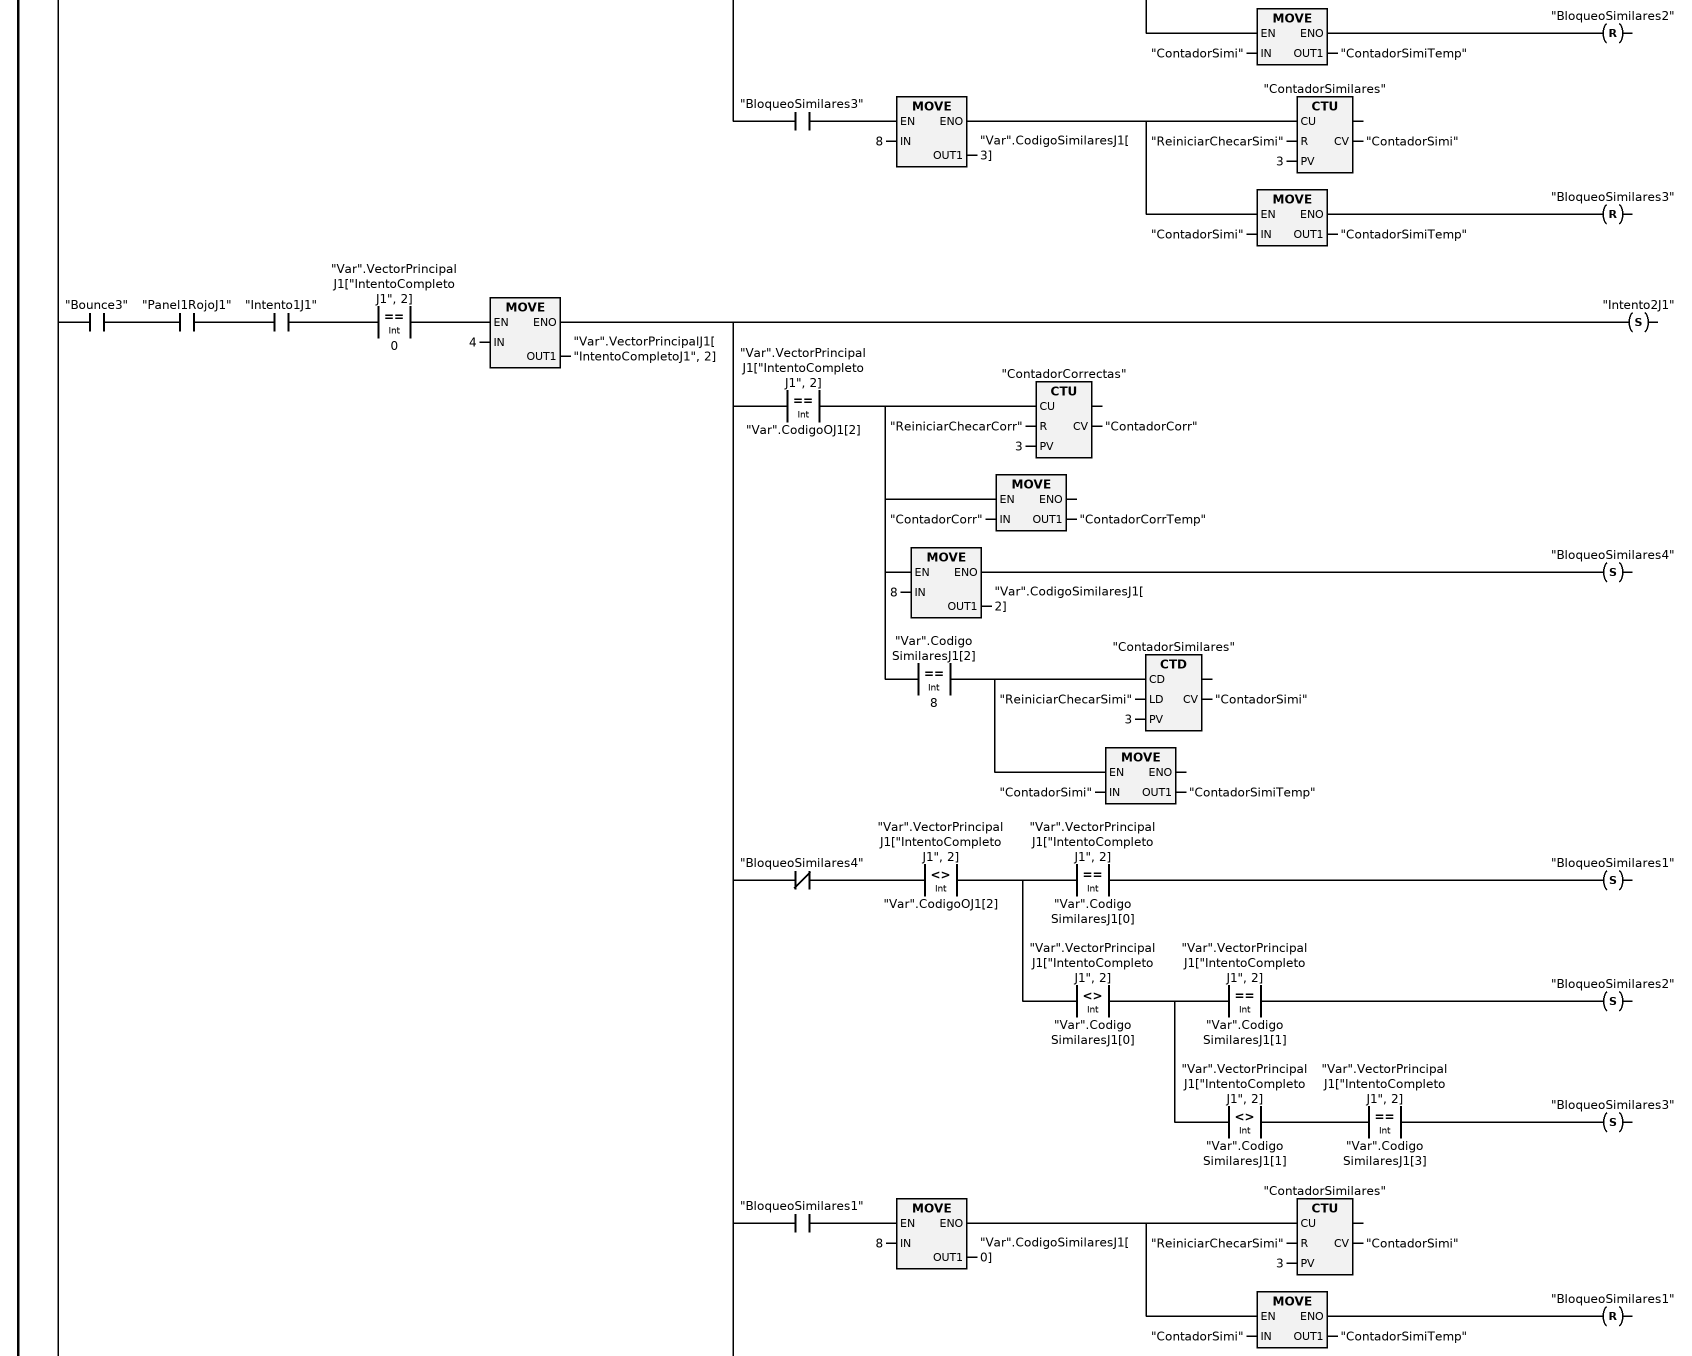
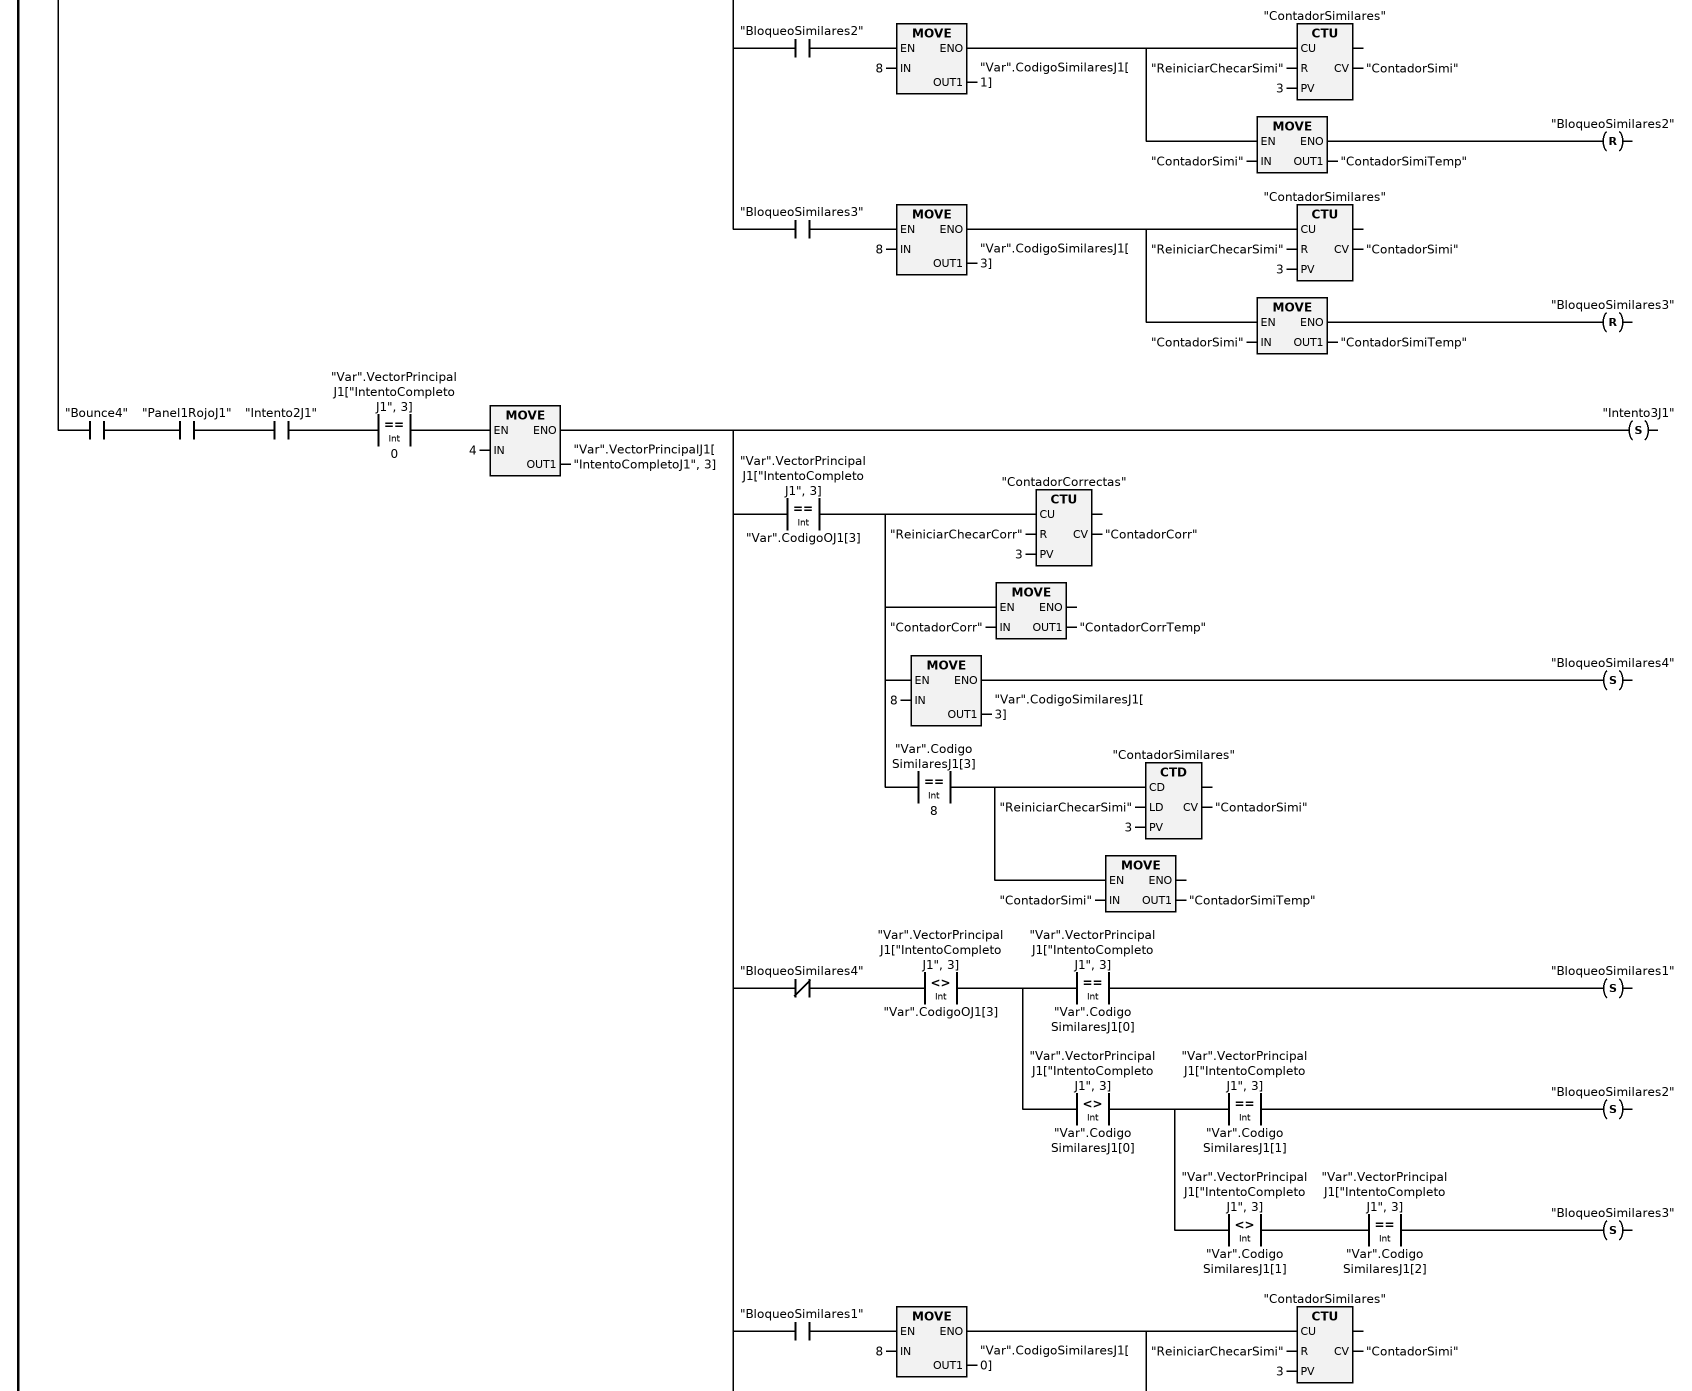
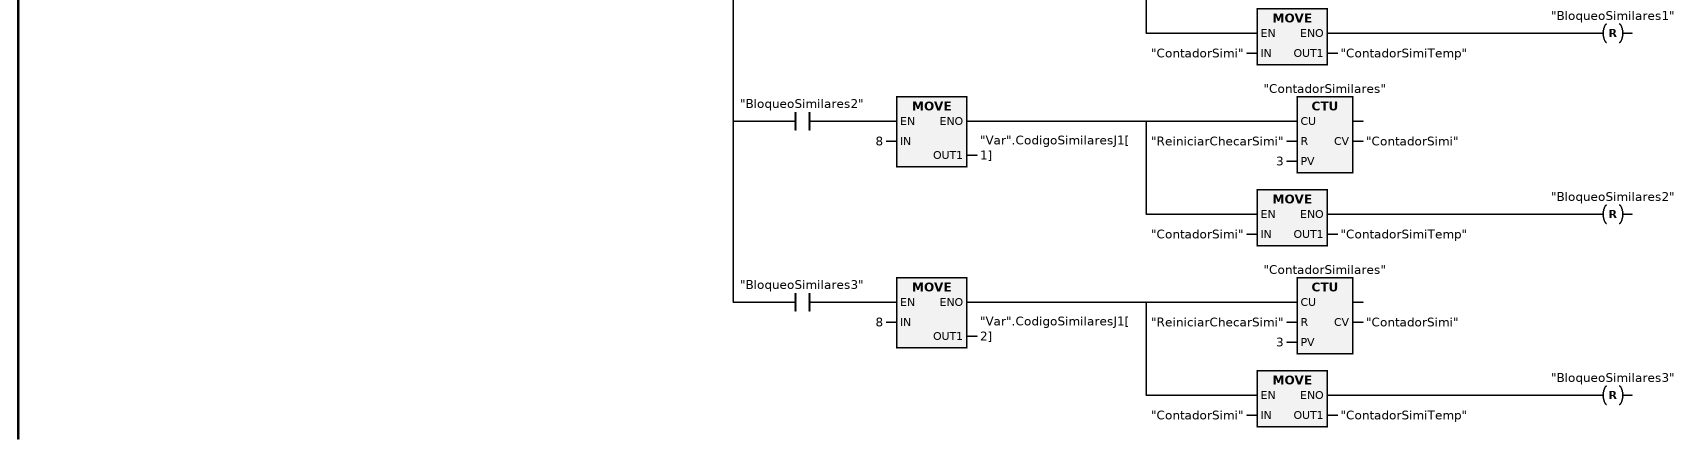
   #_w1 := "Panel1RojoJ1" AND ("Var".VectorPrincipalJ1["IntentoCompletoJ1", 0] = 0) AND "Bounce1";
   IF #_w1 THEN
       "Var".VectorPrincipalJ1["IntentoCompletoJ1", 0] := 4;
       "Var".VectorCorrectas["IntentoCompletoJ1", 0] := 4;
       "Intento0J1" := TRUE;
   END_IF;
   #_w2 := #_w1 AND ("Var".VectorPrincipalJ1["IntentoCompletoJ1", 0] = "Var".CodigoOJ1[0]);
   "ContadorCorrectas".CTU(CU := #_w2, R := "ReiniciarChecarCorr", PV := 3, CV => "ContadorCorr");
   IF #_w2 THEN
       "ContadorCorrTemp" := "ContadorCorr";
       "Var".CodigoSimilaresJ1[0] := 8;
       "BloqueoSimilares4" := TRUE;
   END_IF;
   #_w3 := #_w2 AND ("Var".CodigoSimilaresJ1[0] = 8);
   "ContadorSimilares".CTD(CD := #_w3, LD := "ReiniciarChecarSimi", PV := 3, CV => "ContadorSimi");
   IF #_w3 THEN "ContadorSimiTemp" := "ContadorSimi"; END_IF;
   #_w4 := #_w1 AND NOT "BloqueoSimilares4" AND ("Var".VectorPrincipalJ1["IntentoCompletoJ1", 0] <> "Var".CodigoOJ1[0]);
   IF #_w4 AND ("Var".VectorPrincipalJ1["IntentoCompletoJ1", 0] = "Var".CodigoSimilaresJ1[1]) THEN
       "BloqueoSimilares1" := TRUE;
   END_IF;
   #_w5 := #_w4 AND ("Var".VectorPrincipalJ1["IntentoCompletoJ1", 0] <> "Var".CodigoSimilaresJ1[1]);
   IF #_w5 AND ("Var".VectorPrincipalJ1["IntentoCompletoJ1", 0] = "Var".CodigoSimilaresJ1[2]) THEN
       "BloqueoSimilares2" := TRUE;
   END_IF;
   IF #_w5 AND ("Var".VectorPrincipalJ1["IntentoCompletoJ1", 0] <> "Var".CodigoSimilaresJ1[2]) AND ("Var".VectorPrincipalJ1["IntentoCompletoJ1", 0] = "Var".CodigoSimilaresJ1[3]) THEN
       "BloqueoSimilares3" := TRUE;
   END_IF;
   #_w6 := #_w1 AND "BloqueoSimilares1";
   IF #_w6 THEN "Var".CodigoSimilaresJ1[1] := 8; END_IF;
   "ContadorSimilares".CTU(CU := #_w6, R := "ReiniciarChecarSimi", PV := 3, CV => "ContadorSimi");
   IF #_w6 THEN
       "ContadorSimiTemp" := "ContadorSimi";
       "BloqueoSimilares1" := FALSE;
   END_IF;
   #_w7 := #_w1 AND "BloqueoSimilares2";
   IF #_w7 THEN "Var".CodigoSimilaresJ1[2] := 8; END_IF;
   "ContadorSimilares".CTU(CU := #_w7, R := "ReiniciarChecarSimi", PV := 3, CV => "ContadorSimi");
   IF #_w7 THEN
       "ContadorSimiTemp" := "ContadorSimi";
       "BloqueoSimilares2" := FALSE;
   END_IF;
   #_w8 := #_w1 AND "BloqueoSimilares3";
   IF #_w8 THEN "Var".CodigoSimilaresJ1[3] := 8; END_IF;
   "ContadorSimilares".CTU(CU := #_w8, R := "ReiniciarChecarSimi", PV := 3, CV => "ContadorSimi");
   IF #_w8 THEN
       "ContadorSimiTemp" := "ContadorSimi";
       "BloqueoSimilares3" := FALSE;
   END_IF;
   #_w9 := "Panel1RojoJ1" AND "Bounce2" AND "Panel1RojoJ1" AND "Intento0J1" AND ("Var".VectorPrincipalJ1["IntentoCompletoJ1", 1] = 0);
   IF #_w9 THEN
       "Var".VectorPrincipalJ1["IntentoCompletoJ1", 1] := 4;
       "Intento1J1" := TRUE;
   END_IF;
   #_w10 := #_w9 AND ("Var".VectorPrincipalJ1["IntentoCompletoJ1", 1] = "Var".CodigoOJ1[1]);
   "ContadorCorrectas".CTU(CU := #_w10, R := "ReiniciarChecarCorr", PV := 3, CV => "ContadorCorr");
   IF #_w10 THEN
       "ContadorCorrTemp" := "ContadorCorr";
       "Var".CodigoSimilaresJ1[1] := 8;
       "BloqueoSimilares4" := TRUE;
   END_IF;
   #_w11 := #_w10 AND ("Var".CodigoSimilaresJ1[1] = 8);
   "ContadorSimilares".CTD(CD := #_w11, LD := "ReiniciarChecarSimi", PV := 3, CV => "ContadorSimi");
   IF #_w11 THEN "ContadorSimiTemp" := "ContadorSimi"; END_IF;
   #_w12 := #_w9 AND NOT "BloqueoSimilares4" AND ("Var".VectorPrincipalJ1["IntentoCompletoJ1", 1] <> "Var".CodigoOJ1[1]);
   IF #_w12 AND ("Var".VectorPrincipalJ1["IntentoCompletoJ1", 1] = "Var".CodigoSimilaresJ1[0]) THEN
       "BloqueoSimilares1" := TRUE;
   END_IF;
   #_w13 := #_w12 AND ("Var".VectorPrincipalJ1["IntentoCompletoJ1", 1] <> "Var".CodigoSimilaresJ1[0]);
   IF #_w13 AND ("Var".VectorPrincipalJ1["IntentoCompletoJ1", 1] = "Var".CodigoSimilaresJ1[2]) THEN
       "BloqueoSimilares2" := TRUE;
   END_IF;
   IF #_w13 AND ("Var".VectorPrincipalJ1["IntentoCompletoJ1", 1] <> "Var".CodigoSimilaresJ1[2]) AND ("Var".VectorPrincipalJ1["IntentoCompletoJ1", 1] = "Var".CodigoSimilaresJ1[3]) THEN
       "BloqueoSimilares3" := TRUE;
   END_IF;
   #_w14 := #_w9 AND "BloqueoSimilares1";
   IF #_w14 THEN "Var".CodigoSimilaresJ1[0] := 8; END_IF;
   "ContadorSimilares".CTU(CU := #_w14, R := "ReiniciarChecarSimi", PV := 3, CV => "ContadorSimi");
   IF #_w14 THEN
       "ContadorSimiTemp" := "ContadorSimi";
       "BloqueoSimilares1" := FALSE;
   END_IF;
   #_w15 := #_w9 AND "BloqueoSimilares2";
   IF #_w15 THEN "Var".CodigoSimilaresJ1[2] := 8; END_IF;
   "ContadorSimilares".CTU(CU := #_w15, R := "ReiniciarChecarSimi", PV := 3, CV => "ContadorSimi");
   IF #_w15 THEN
       "ContadorSimiTemp" := "ContadorSimi";
       "BloqueoSimilares2" := FALSE;
   END_IF;
   #_w16 := #_w9 AND "BloqueoSimilares3";
   IF #_w16 THEN "Var".CodigoSimilaresJ1[3] := 8; END_IF;
   "ContadorSimilares".CTU(CU := #_w16, R := "ReiniciarChecarSimi", PV := 3, CV => "ContadorSimi");
   IF #_w16 THEN
       "ContadorSimiTemp" := "ContadorSimi";
       "BloqueoSimilares3" := FALSE;
   END_IF;
   #_w17 := "Panel1RojoJ1" AND "Bounce3" AND "Panel1RojoJ1" AND "Intento1J1" AND ("Var".VectorPrincipalJ1["IntentoCompletoJ1", 2] = 0);
   IF #_w17 THEN
       "Var".VectorPrincipalJ1["IntentoCompletoJ1", 2] := 4;
       "Intento2J1" := TRUE;
   END_IF;
   #_w18 := #_w17 AND ("Var".VectorPrincipalJ1["IntentoCompletoJ1", 2] = "Var".CodigoOJ1[2]);
   "ContadorCorrectas".CTU(CU := #_w18, R := "ReiniciarChecarCorr", PV := 3, CV => "ContadorCorr");
   IF #_w18 THEN
       "ContadorCorrTemp" := "ContadorCorr";
       "Var".CodigoSimilaresJ1[2] := 8;
       "BloqueoSimilares4" := TRUE;
   END_IF;
   #_w19 := #_w18 AND ("Var".CodigoSimilaresJ1[2] = 8);
   "ContadorSimilares".CTD(CD := #_w19, LD := "ReiniciarChecarSimi", PV := 3, CV => "ContadorSimi");
   IF #_w19 THEN "ContadorSimiTemp" := "ContadorSimi"; END_IF;
   #_w20 := #_w17 AND NOT "BloqueoSimilares4" AND ("Var".VectorPrincipalJ1["IntentoCompletoJ1", 2] <> "Var".CodigoOJ1[2]);
   IF #_w20 AND ("Var".VectorPrincipalJ1["IntentoCompletoJ1", 2] = "Var".CodigoSimilaresJ1[0]) THEN
       "BloqueoSimilares1" := TRUE;
   END_IF;
   #_w21 := #_w20 AND ("Var".VectorPrincipalJ1["IntentoCompletoJ1", 2] <> "Var".CodigoSimilaresJ1[0]);
   IF #_w21 AND ("Var".VectorPrincipalJ1["IntentoCompletoJ1", 2] = "Var".CodigoSimilaresJ1[1]) THEN
       "BloqueoSimilares2" := TRUE;
   END_IF;
   IF #_w21 AND ("Var".VectorPrincipalJ1["IntentoCompletoJ1", 2] <> "Var".CodigoSimilaresJ1[1]) AND ("Var".VectorPrincipalJ1["IntentoCompletoJ1", 2] = "Var".CodigoSimilaresJ1[3]) THEN
       "BloqueoSimilares3" := TRUE;
   END_IF;
   #_w22 := #_w17 AND "BloqueoSimilares1";
   IF #_w22 THEN "Var".CodigoSimilaresJ1[0] := 8; END_IF;
   "ContadorSimilares".CTU(CU := #_w22, R := "ReiniciarChecarSimi", PV := 3, CV => "ContadorSimi");
   IF #_w22 THEN
       "ContadorSimiTemp" := "ContadorSimi";
       "BloqueoSimilares1" := FALSE;
   END_IF;
   #_w23 := #_w17 AND "BloqueoSimilares2";
   IF #_w23 THEN "Var".CodigoSimilaresJ1[1] := 8; END_IF;
   "ContadorSimilares".CTU(CU := #_w23, R := "ReiniciarChecarSimi", PV := 3, CV => "ContadorSimi");
   IF #_w23 THEN
       "ContadorSimiTemp" := "ContadorSimi";
       "BloqueoSimilares2" := FALSE;
   END_IF;
   #_w24 := #_w17 AND "BloqueoSimilares3";
   IF #_w24 THEN "Var".CodigoSimilaresJ1[3] := 8; END_IF;
   "ContadorSimilares".CTU(CU := #_w24, R := "ReiniciarChecarSimi", PV := 3, CV => "ContadorSimi");
   IF #_w24 THEN
       "ContadorSimiTemp" := "ContadorSimi";
       "BloqueoSimilares3" := FALSE;
   END_IF;
   #_w25 := "Panel1RojoJ1" AND "Bounce4" AND "Panel1RojoJ1" AND "Intento2J1" AND ("Var".VectorPrincipalJ1["IntentoCompletoJ1", 3] = 0);
   IF #_w25 THEN
       "Var".VectorPrincipalJ1["IntentoCompletoJ1", 3] := 4;
       "Intento3J1" := TRUE;
   END_IF;
   #_w26 := #_w25 AND ("Var".VectorPrincipalJ1["IntentoCompletoJ1", 3] = "Var".CodigoOJ1[3]);
   "ContadorCorrectas".CTU(CU := #_w26, R := "ReiniciarChecarCorr", PV := 3, CV => "ContadorCorr");
   IF #_w26 THEN
       "ContadorCorrTemp" := "ContadorCorr";
       "Var".CodigoSimilaresJ1[3] := 8;
       "BloqueoSimilares4" := TRUE;
   END_IF;
   #_w27 := #_w26 AND ("Var".CodigoSimilaresJ1[3] = 8);
   "ContadorSimilares".CTD(CD := #_w27, LD := "ReiniciarChecarSimi", PV := 3, CV => "ContadorSimi");
   IF #_w27 THEN "ContadorSimiTemp" := "ContadorSimi"; END_IF;
   #_w28 := #_w25 AND NOT "BloqueoSimilares4" AND ("Var".VectorPrincipalJ1["IntentoCompletoJ1", 3] <> "Var".CodigoOJ1[3]);
   IF #_w28 AND ("Var".VectorPrincipalJ1["IntentoCompletoJ1", 3] = "Var".CodigoSimilaresJ1[0]) THEN
       "BloqueoSimilares1" := TRUE;
   END_IF;
   #_w29 := #_w28 AND ("Var".VectorPrincipalJ1["IntentoCompletoJ1", 3] <> "Var".CodigoSimilaresJ1[0]);
   IF #_w29 AND ("Var".VectorPrincipalJ1["IntentoCompletoJ1", 3] = "Var".CodigoSimilaresJ1[1]) THEN
       "BloqueoSimilares2" := TRUE;
   END_IF;
   IF #_w29 AND ("Var".VectorPrincipalJ1["IntentoCompletoJ1", 3] <> "Var".CodigoSimilaresJ1[1]) AND ("Var".VectorPrincipalJ1["IntentoCompletoJ1", 3] = "Var".CodigoSimilaresJ1[2]) THEN
       "BloqueoSimilares3" := TRUE;
   END_IF;
   #_w30 := #_w25 AND "BloqueoSimilares1";
   IF #_w30 THEN "Var".CodigoSimilaresJ1[0] := 8; END_IF;
   "ContadorSimilares".CTU(CU := #_w30, R := "ReiniciarChecarSimi", PV := 3, CV => "ContadorSimi");
   IF #_w30 THEN
       "ContadorSimiTemp" := "ContadorSimi";
       "BloqueoSimilares1" := FALSE;
   END_IF;
   #_w31 := #_w25 AND "BloqueoSimilares2";
   IF #_w31 THEN "Var".CodigoSimilaresJ1[1] := 8; END_IF;
   "ContadorSimilares".CTU(CU := #_w31, R := "ReiniciarChecarSimi", PV := 3, CV => "ContadorSimi");
   IF #_w31 THEN
       "ContadorSimiTemp" := "ContadorSimi";
       "BloqueoSimilares2" := FALSE;
   END_IF;
   #_w32 := #_w25 AND "BloqueoSimilares3";
   IF #_w32 THEN "Var".CodigoSimilaresJ1[2] := 8; END_IF;
   "ContadorSimilares".CTU(CU := #_w32, R := "ReiniciarChecarSimi", PV := 3, CV => "ContadorSimi");
   IF #_w32 THEN
       "ContadorSimiTemp" := "ContadorSimi";
       "BloqueoSimilares3" := FALSE;
   END_IF;
END_REGION

REGION Network 10: Azul
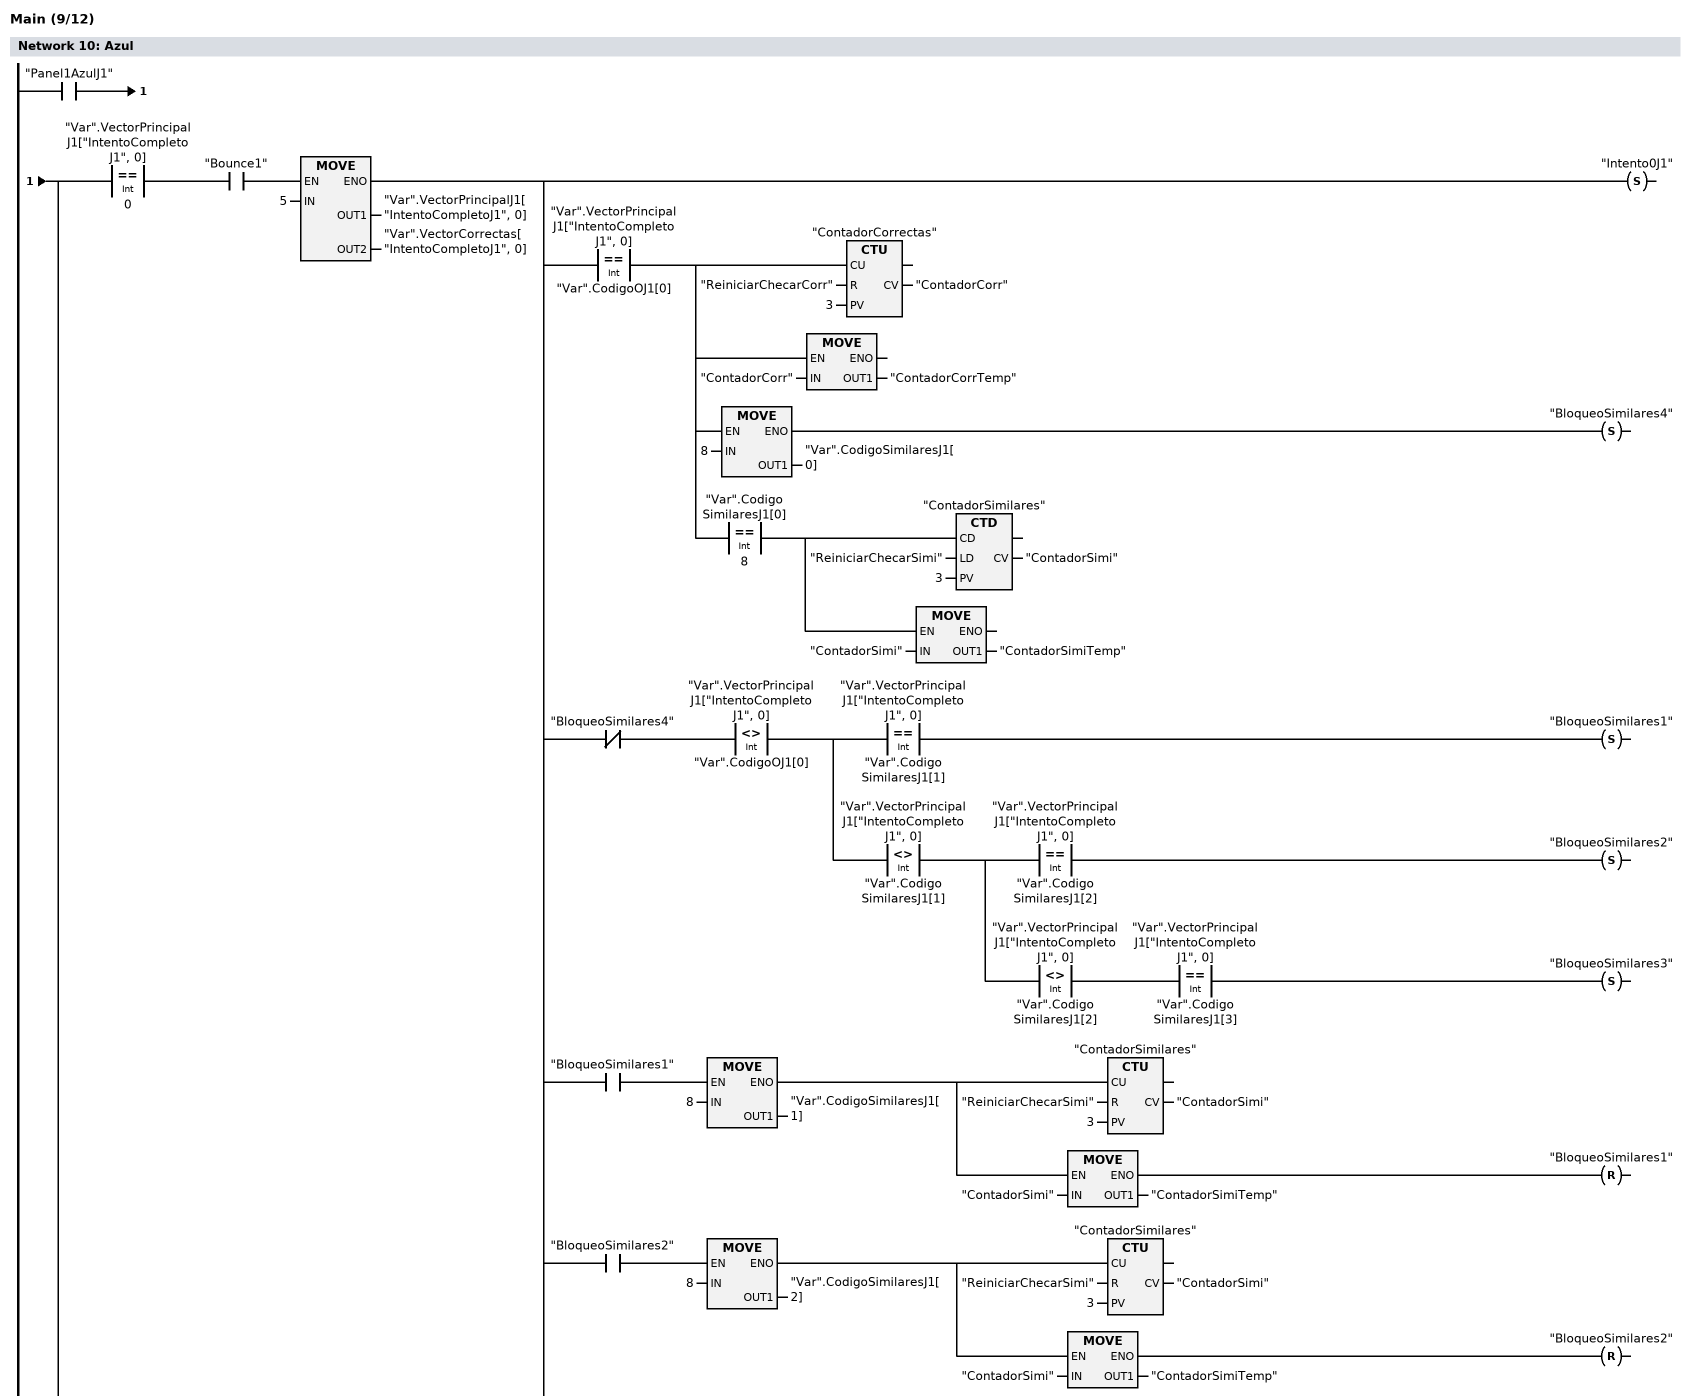
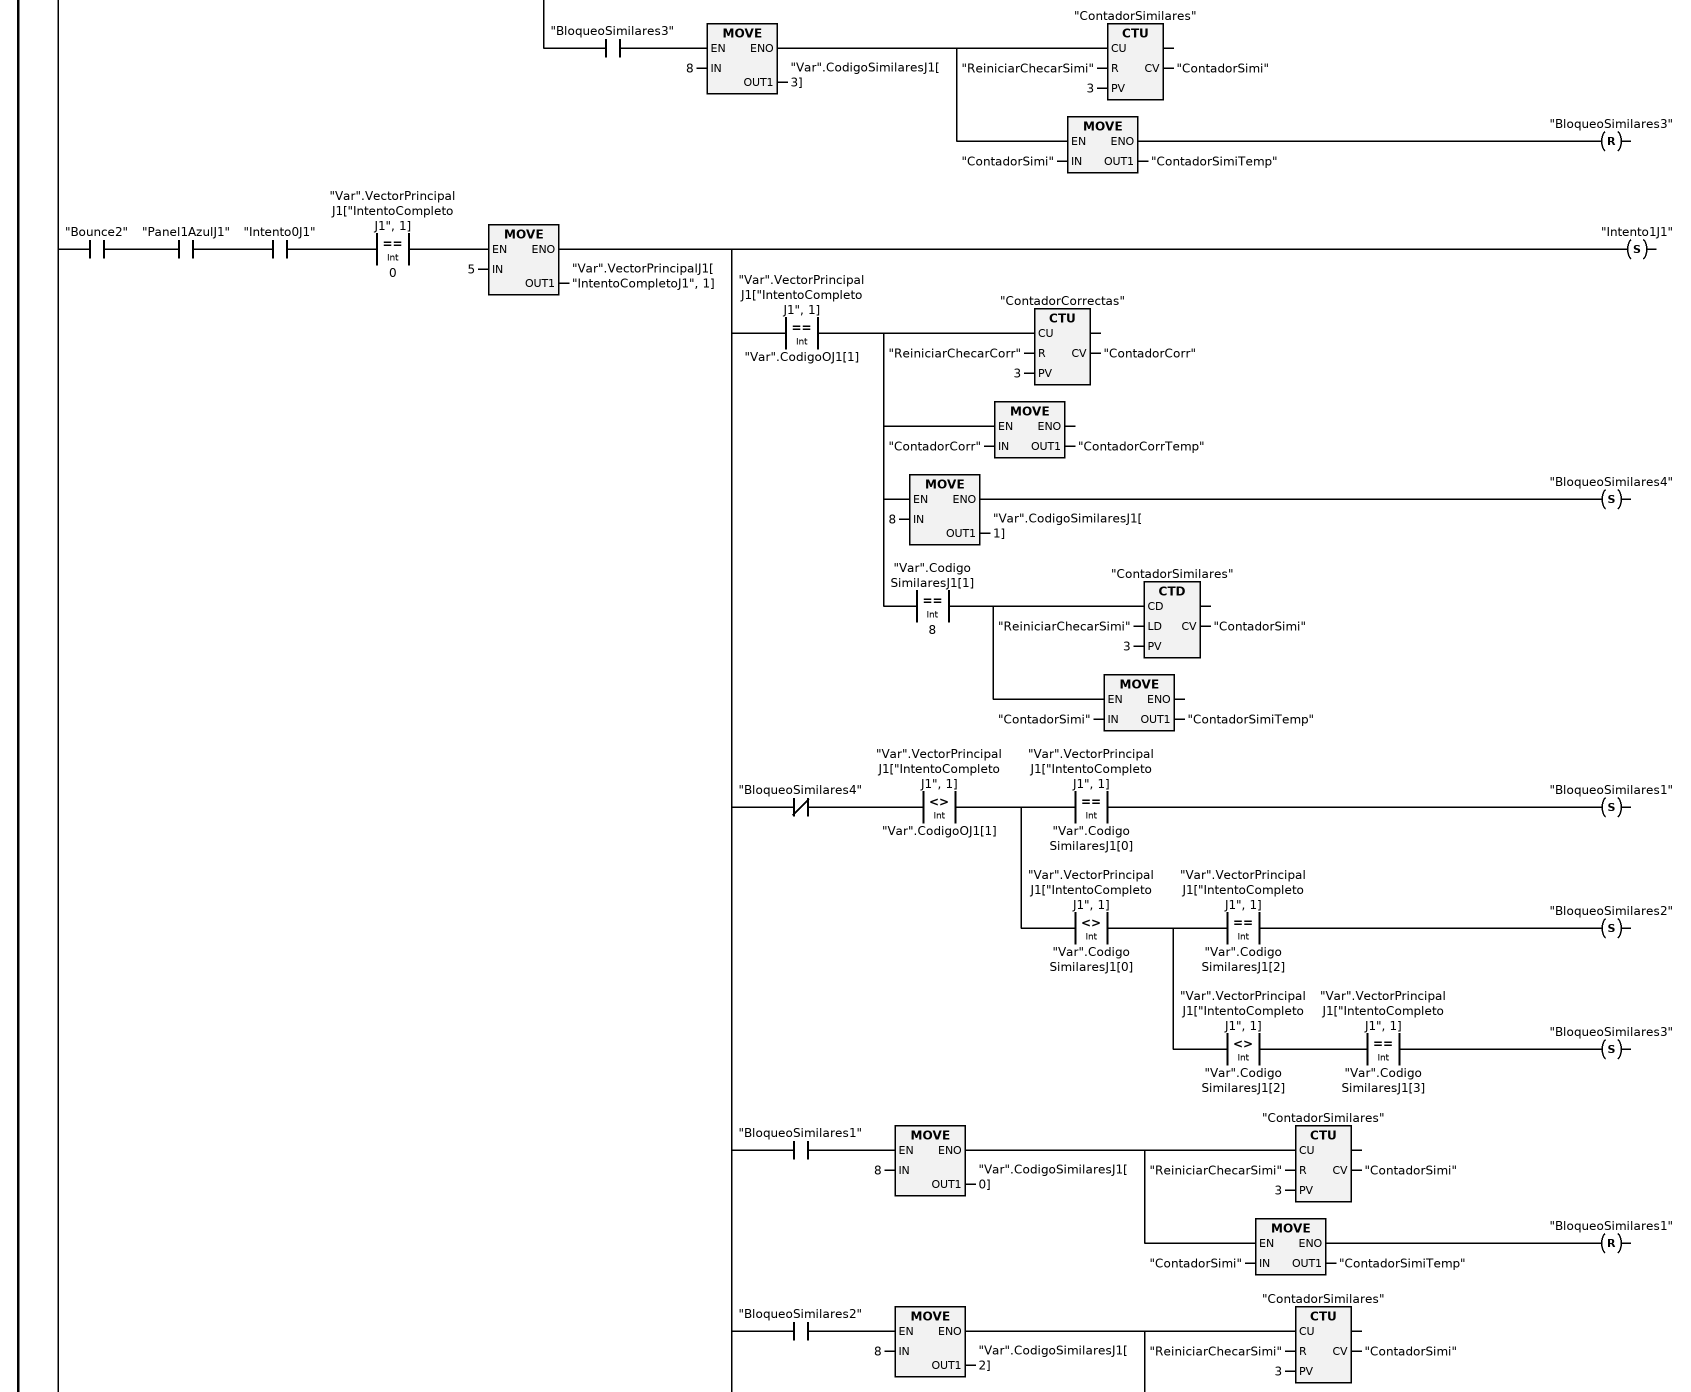
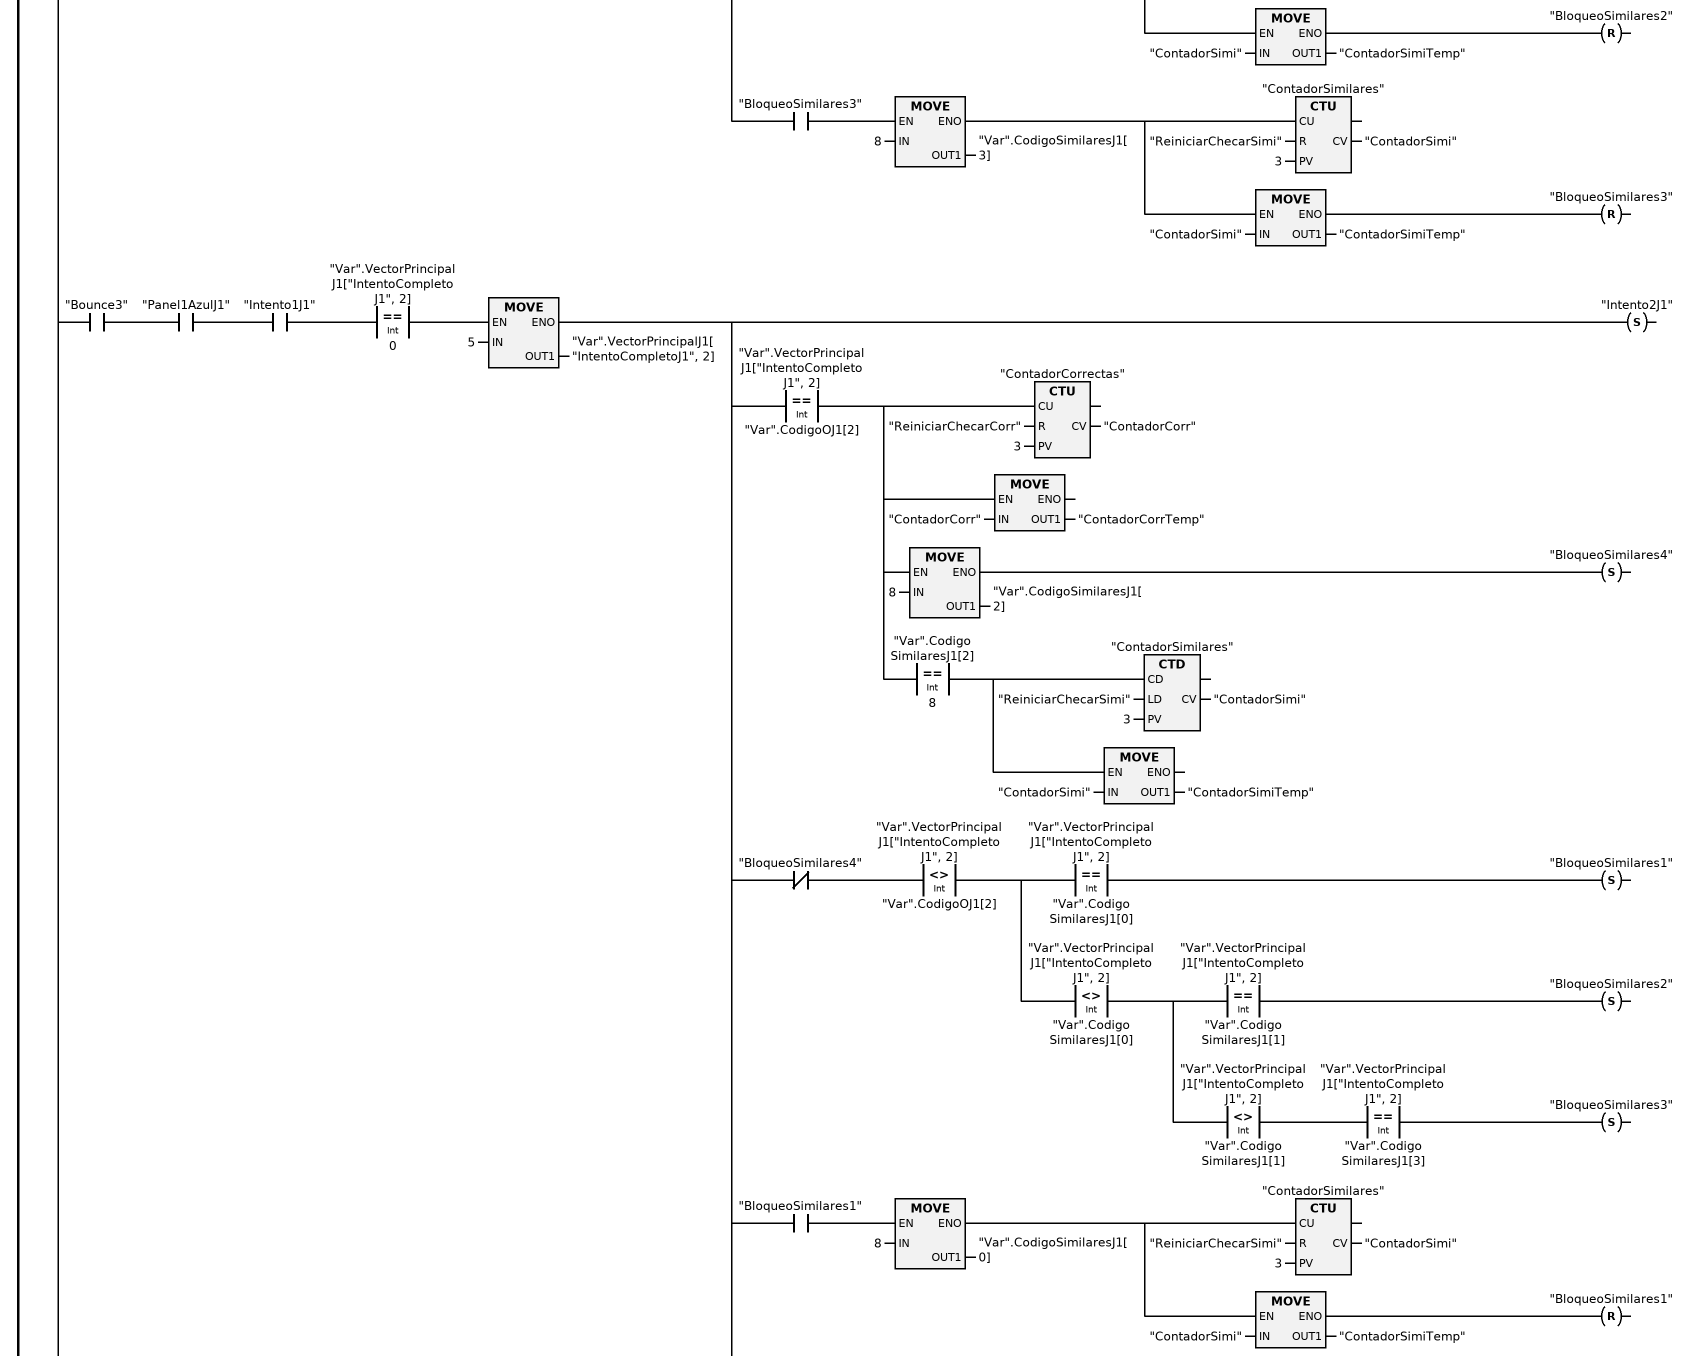
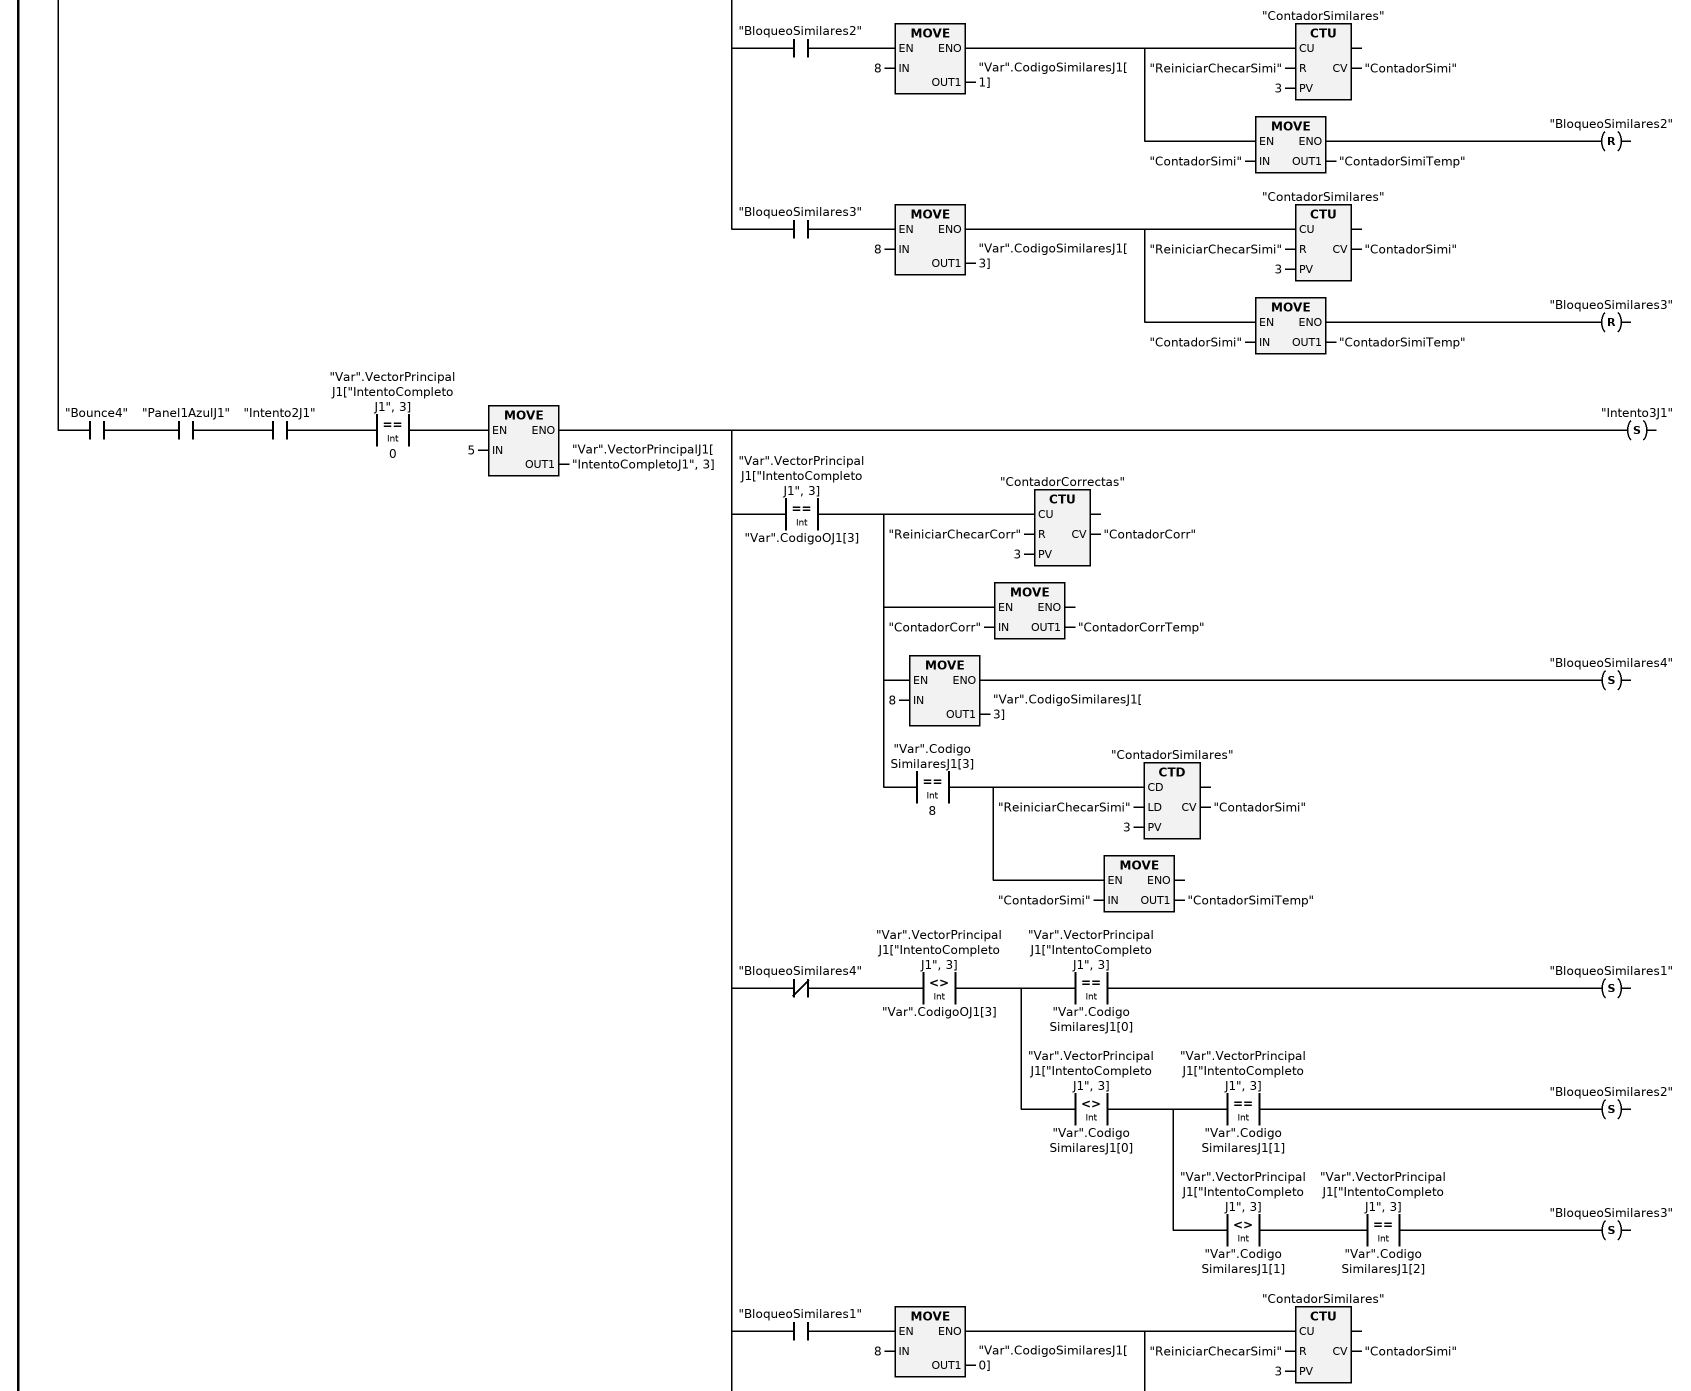
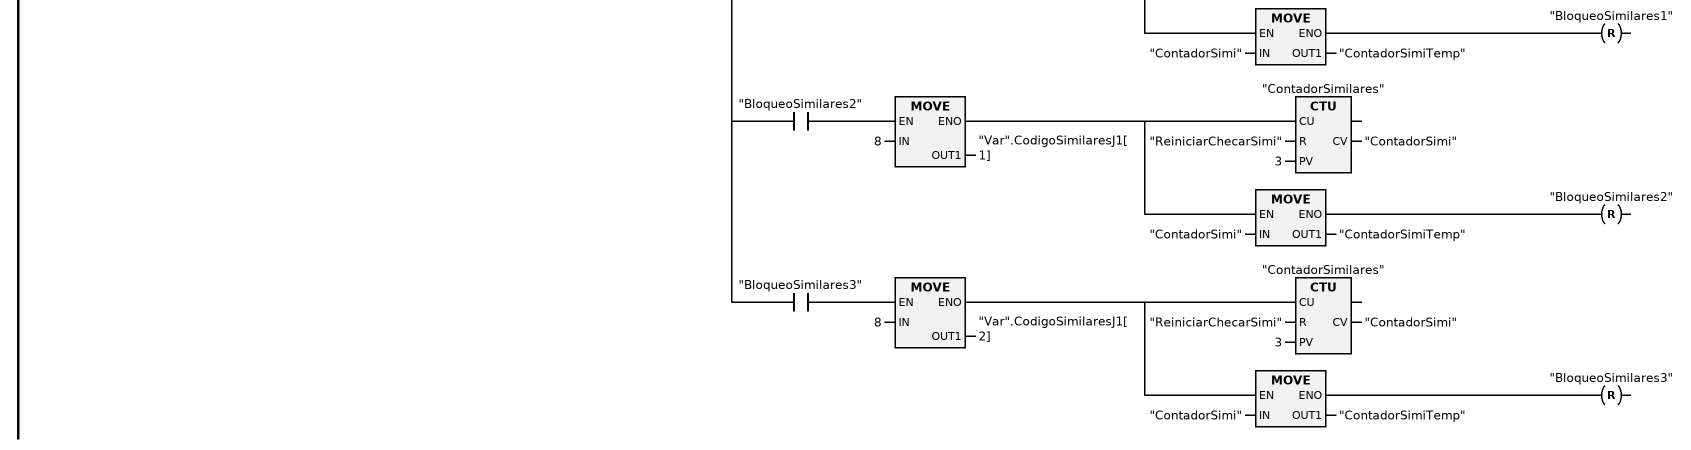
   #_w1 := "Panel1AzulJ1" AND ("Var".VectorPrincipalJ1["IntentoCompletoJ1", 0] = 0) AND "Bounce1";
   IF #_w1 THEN
       "Var".VectorPrincipalJ1["IntentoCompletoJ1", 0] := 5;
       "Var".VectorCorrectas["IntentoCompletoJ1", 0] := 5;
       "Intento0J1" := TRUE;
   END_IF;
   #_w2 := #_w1 AND ("Var".VectorPrincipalJ1["IntentoCompletoJ1", 0] = "Var".CodigoOJ1[0]);
   "ContadorCorrectas".CTU(CU := #_w2, R := "ReiniciarChecarCorr", PV := 3, CV => "ContadorCorr");
   IF #_w2 THEN
       "ContadorCorrTemp" := "ContadorCorr";
       "Var".CodigoSimilaresJ1[0] := 8;
       "BloqueoSimilares4" := TRUE;
   END_IF;
   #_w3 := #_w2 AND ("Var".CodigoSimilaresJ1[0] = 8);
   "ContadorSimilares".CTD(CD := #_w3, LD := "ReiniciarChecarSimi", PV := 3, CV => "ContadorSimi");
   IF #_w3 THEN "ContadorSimiTemp" := "ContadorSimi"; END_IF;
   #_w4 := #_w1 AND NOT "BloqueoSimilares4" AND ("Var".VectorPrincipalJ1["IntentoCompletoJ1", 0] <> "Var".CodigoOJ1[0]);
   IF #_w4 AND ("Var".VectorPrincipalJ1["IntentoCompletoJ1", 0] = "Var".CodigoSimilaresJ1[1]) THEN
       "BloqueoSimilares1" := TRUE;
   END_IF;
   #_w5 := #_w4 AND ("Var".VectorPrincipalJ1["IntentoCompletoJ1", 0] <> "Var".CodigoSimilaresJ1[1]);
   IF #_w5 AND ("Var".VectorPrincipalJ1["IntentoCompletoJ1", 0] = "Var".CodigoSimilaresJ1[2]) THEN
       "BloqueoSimilares2" := TRUE;
   END_IF;
   IF #_w5 AND ("Var".VectorPrincipalJ1["IntentoCompletoJ1", 0] <> "Var".CodigoSimilaresJ1[2]) AND ("Var".VectorPrincipalJ1["IntentoCompletoJ1", 0] = "Var".CodigoSimilaresJ1[3]) THEN
       "BloqueoSimilares3" := TRUE;
   END_IF;
   #_w6 := #_w1 AND "BloqueoSimilares1";
   IF #_w6 THEN "Var".CodigoSimilaresJ1[1] := 8; END_IF;
   "ContadorSimilares".CTU(CU := #_w6, R := "ReiniciarChecarSimi", PV := 3, CV => "ContadorSimi");
   IF #_w6 THEN
       "ContadorSimiTemp" := "ContadorSimi";
       "BloqueoSimilares1" := FALSE;
   END_IF;
   #_w7 := #_w1 AND "BloqueoSimilares2";
   IF #_w7 THEN "Var".CodigoSimilaresJ1[2] := 8; END_IF;
   "ContadorSimilares".CTU(CU := #_w7, R := "ReiniciarChecarSimi", PV := 3, CV => "ContadorSimi");
   IF #_w7 THEN
       "ContadorSimiTemp" := "ContadorSimi";
       "BloqueoSimilares2" := FALSE;
   END_IF;
   #_w8 := #_w1 AND "BloqueoSimilares3";
   IF #_w8 THEN "Var".CodigoSimilaresJ1[3] := 8; END_IF;
   "ContadorSimilares".CTU(CU := #_w8, R := "ReiniciarChecarSimi", PV := 3, CV => "ContadorSimi");
   IF #_w8 THEN
       "ContadorSimiTemp" := "ContadorSimi";
       "BloqueoSimilares3" := FALSE;
   END_IF;
   #_w9 := "Panel1AzulJ1" AND "Bounce2" AND "Panel1AzulJ1" AND "Intento0J1" AND ("Var".VectorPrincipalJ1["IntentoCompletoJ1", 1] = 0);
   IF #_w9 THEN
       "Var".VectorPrincipalJ1["IntentoCompletoJ1", 1] := 5;
       "Intento1J1" := TRUE;
   END_IF;
   #_w10 := #_w9 AND ("Var".VectorPrincipalJ1["IntentoCompletoJ1", 1] = "Var".CodigoOJ1[1]);
   "ContadorCorrectas".CTU(CU := #_w10, R := "ReiniciarChecarCorr", PV := 3, CV => "ContadorCorr");
   IF #_w10 THEN
       "ContadorCorrTemp" := "ContadorCorr";
       "Var".CodigoSimilaresJ1[1] := 8;
       "BloqueoSimilares4" := TRUE;
   END_IF;
   #_w11 := #_w10 AND ("Var".CodigoSimilaresJ1[1] = 8);
   "ContadorSimilares".CTD(CD := #_w11, LD := "ReiniciarChecarSimi", PV := 3, CV => "ContadorSimi");
   IF #_w11 THEN "ContadorSimiTemp" := "ContadorSimi"; END_IF;
   #_w12 := #_w9 AND NOT "BloqueoSimilares4" AND ("Var".VectorPrincipalJ1["IntentoCompletoJ1", 1] <> "Var".CodigoOJ1[1]);
   IF #_w12 AND ("Var".VectorPrincipalJ1["IntentoCompletoJ1", 1] = "Var".CodigoSimilaresJ1[0]) THEN
       "BloqueoSimilares1" := TRUE;
   END_IF;
   #_w13 := #_w12 AND ("Var".VectorPrincipalJ1["IntentoCompletoJ1", 1] <> "Var".CodigoSimilaresJ1[0]);
   IF #_w13 AND ("Var".VectorPrincipalJ1["IntentoCompletoJ1", 1] = "Var".CodigoSimilaresJ1[2]) THEN
       "BloqueoSimilares2" := TRUE;
   END_IF;
   IF #_w13 AND ("Var".VectorPrincipalJ1["IntentoCompletoJ1", 1] <> "Var".CodigoSimilaresJ1[2]) AND ("Var".VectorPrincipalJ1["IntentoCompletoJ1", 1] = "Var".CodigoSimilaresJ1[3]) THEN
       "BloqueoSimilares3" := TRUE;
   END_IF;
   #_w14 := #_w9 AND "BloqueoSimilares1";
   IF #_w14 THEN "Var".CodigoSimilaresJ1[0] := 8; END_IF;
   "ContadorSimilares".CTU(CU := #_w14, R := "ReiniciarChecarSimi", PV := 3, CV => "ContadorSimi");
   IF #_w14 THEN
       "ContadorSimiTemp" := "ContadorSimi";
       "BloqueoSimilares1" := FALSE;
   END_IF;
   #_w15 := #_w9 AND "BloqueoSimilares2";
   IF #_w15 THEN "Var".CodigoSimilaresJ1[2] := 8; END_IF;
   "ContadorSimilares".CTU(CU := #_w15, R := "ReiniciarChecarSimi", PV := 3, CV => "ContadorSimi");
   IF #_w15 THEN
       "ContadorSimiTemp" := "ContadorSimi";
       "BloqueoSimilares2" := FALSE;
   END_IF;
   #_w16 := #_w9 AND "BloqueoSimilares3";
   IF #_w16 THEN "Var".CodigoSimilaresJ1[3] := 8; END_IF;
   "ContadorSimilares".CTU(CU := #_w16, R := "ReiniciarChecarSimi", PV := 3, CV => "ContadorSimi");
   IF #_w16 THEN
       "ContadorSimiTemp" := "ContadorSimi";
       "BloqueoSimilares3" := FALSE;
   END_IF;
   #_w17 := "Panel1AzulJ1" AND "Bounce3" AND "Panel1AzulJ1" AND "Intento1J1" AND ("Var".VectorPrincipalJ1["IntentoCompletoJ1", 2] = 0);
   IF #_w17 THEN
       "Var".VectorPrincipalJ1["IntentoCompletoJ1", 2] := 5;
       "Intento2J1" := TRUE;
   END_IF;
   #_w18 := #_w17 AND ("Var".VectorPrincipalJ1["IntentoCompletoJ1", 2] = "Var".CodigoOJ1[2]);
   "ContadorCorrectas".CTU(CU := #_w18, R := "ReiniciarChecarCorr", PV := 3, CV => "ContadorCorr");
   IF #_w18 THEN
       "ContadorCorrTemp" := "ContadorCorr";
       "Var".CodigoSimilaresJ1[2] := 8;
       "BloqueoSimilares4" := TRUE;
   END_IF;
   #_w19 := #_w18 AND ("Var".CodigoSimilaresJ1[2] = 8);
   "ContadorSimilares".CTD(CD := #_w19, LD := "ReiniciarChecarSimi", PV := 3, CV => "ContadorSimi");
   IF #_w19 THEN "ContadorSimiTemp" := "ContadorSimi"; END_IF;
   #_w20 := #_w17 AND NOT "BloqueoSimilares4" AND ("Var".VectorPrincipalJ1["IntentoCompletoJ1", 2] <> "Var".CodigoOJ1[2]);
   IF #_w20 AND ("Var".VectorPrincipalJ1["IntentoCompletoJ1", 2] = "Var".CodigoSimilaresJ1[0]) THEN
       "BloqueoSimilares1" := TRUE;
   END_IF;
   #_w21 := #_w20 AND ("Var".VectorPrincipalJ1["IntentoCompletoJ1", 2] <> "Var".CodigoSimilaresJ1[0]);
   IF #_w21 AND ("Var".VectorPrincipalJ1["IntentoCompletoJ1", 2] = "Var".CodigoSimilaresJ1[1]) THEN
       "BloqueoSimilares2" := TRUE;
   END_IF;
   IF #_w21 AND ("Var".VectorPrincipalJ1["IntentoCompletoJ1", 2] <> "Var".CodigoSimilaresJ1[1]) AND ("Var".VectorPrincipalJ1["IntentoCompletoJ1", 2] = "Var".CodigoSimilaresJ1[3]) THEN
       "BloqueoSimilares3" := TRUE;
   END_IF;
   #_w22 := #_w17 AND "BloqueoSimilares1";
   IF #_w22 THEN "Var".CodigoSimilaresJ1[0] := 8; END_IF;
   "ContadorSimilares".CTU(CU := #_w22, R := "ReiniciarChecarSimi", PV := 3, CV => "ContadorSimi");
   IF #_w22 THEN
       "ContadorSimiTemp" := "ContadorSimi";
       "BloqueoSimilares1" := FALSE;
   END_IF;
   #_w23 := #_w17 AND "BloqueoSimilares2";
   IF #_w23 THEN "Var".CodigoSimilaresJ1[1] := 8; END_IF;
   "ContadorSimilares".CTU(CU := #_w23, R := "ReiniciarChecarSimi", PV := 3, CV => "ContadorSimi");
   IF #_w23 THEN
       "ContadorSimiTemp" := "ContadorSimi";
       "BloqueoSimilares2" := FALSE;
   END_IF;
   #_w24 := #_w17 AND "BloqueoSimilares3";
   IF #_w24 THEN "Var".CodigoSimilaresJ1[3] := 8; END_IF;
   "ContadorSimilares".CTU(CU := #_w24, R := "ReiniciarChecarSimi", PV := 3, CV => "ContadorSimi");
   IF #_w24 THEN
       "ContadorSimiTemp" := "ContadorSimi";
       "BloqueoSimilares3" := FALSE;
   END_IF;
   #_w25 := "Panel1AzulJ1" AND "Bounce4" AND "Panel1AzulJ1" AND "Intento2J1" AND ("Var".VectorPrincipalJ1["IntentoCompletoJ1", 3] = 0);
   IF #_w25 THEN
       "Var".VectorPrincipalJ1["IntentoCompletoJ1", 3] := 5;
       "Intento3J1" := TRUE;
   END_IF;
   #_w26 := #_w25 AND ("Var".VectorPrincipalJ1["IntentoCompletoJ1", 3] = "Var".CodigoOJ1[3]);
   "ContadorCorrectas".CTU(CU := #_w26, R := "ReiniciarChecarCorr", PV := 3, CV => "ContadorCorr");
   IF #_w26 THEN
       "ContadorCorrTemp" := "ContadorCorr";
       "Var".CodigoSimilaresJ1[3] := 8;
       "BloqueoSimilares4" := TRUE;
   END_IF;
   #_w27 := #_w26 AND ("Var".CodigoSimilaresJ1[3] = 8);
   "ContadorSimilares".CTD(CD := #_w27, LD := "ReiniciarChecarSimi", PV := 3, CV => "ContadorSimi");
   IF #_w27 THEN "ContadorSimiTemp" := "ContadorSimi"; END_IF;
   #_w28 := #_w25 AND NOT "BloqueoSimilares4" AND ("Var".VectorPrincipalJ1["IntentoCompletoJ1", 3] <> "Var".CodigoOJ1[3]);
   IF #_w28 AND ("Var".VectorPrincipalJ1["IntentoCompletoJ1", 3] = "Var".CodigoSimilaresJ1[0]) THEN
       "BloqueoSimilares1" := TRUE;
   END_IF;
   #_w29 := #_w28 AND ("Var".VectorPrincipalJ1["IntentoCompletoJ1", 3] <> "Var".CodigoSimilaresJ1[0]);
   IF #_w29 AND ("Var".VectorPrincipalJ1["IntentoCompletoJ1", 3] = "Var".CodigoSimilaresJ1[1]) THEN
       "BloqueoSimilares2" := TRUE;
   END_IF;
   IF #_w29 AND ("Var".VectorPrincipalJ1["IntentoCompletoJ1", 3] <> "Var".CodigoSimilaresJ1[1]) AND ("Var".VectorPrincipalJ1["IntentoCompletoJ1", 3] = "Var".CodigoSimilaresJ1[2]) THEN
       "BloqueoSimilares3" := TRUE;
   END_IF;
   #_w30 := #_w25 AND "BloqueoSimilares1";
   IF #_w30 THEN "Var".CodigoSimilaresJ1[0] := 8; END_IF;
   "ContadorSimilares".CTU(CU := #_w30, R := "ReiniciarChecarSimi", PV := 3, CV => "ContadorSimi");
   IF #_w30 THEN
       "ContadorSimiTemp" := "ContadorSimi";
       "BloqueoSimilares1" := FALSE;
   END_IF;
   #_w31 := #_w25 AND "BloqueoSimilares2";
   IF #_w31 THEN "Var".CodigoSimilaresJ1[1] := 8; END_IF;
   "ContadorSimilares".CTU(CU := #_w31, R := "ReiniciarChecarSimi", PV := 3, CV => "ContadorSimi");
   IF #_w31 THEN
       "ContadorSimiTemp" := "ContadorSimi";
       "BloqueoSimilares2" := FALSE;
   END_IF;
   #_w32 := #_w25 AND "BloqueoSimilares3";
   IF #_w32 THEN "Var".CodigoSimilaresJ1[2] := 8; END_IF;
   "ContadorSimilares".CTU(CU := #_w32, R := "ReiniciarChecarSimi", PV := 3, CV => "ContadorSimi");
   IF #_w32 THEN
       "ContadorSimiTemp" := "ContadorSimi";
       "BloqueoSimilares3" := FALSE;
   END_IF;
END_REGION

REGION Network 11: Verde
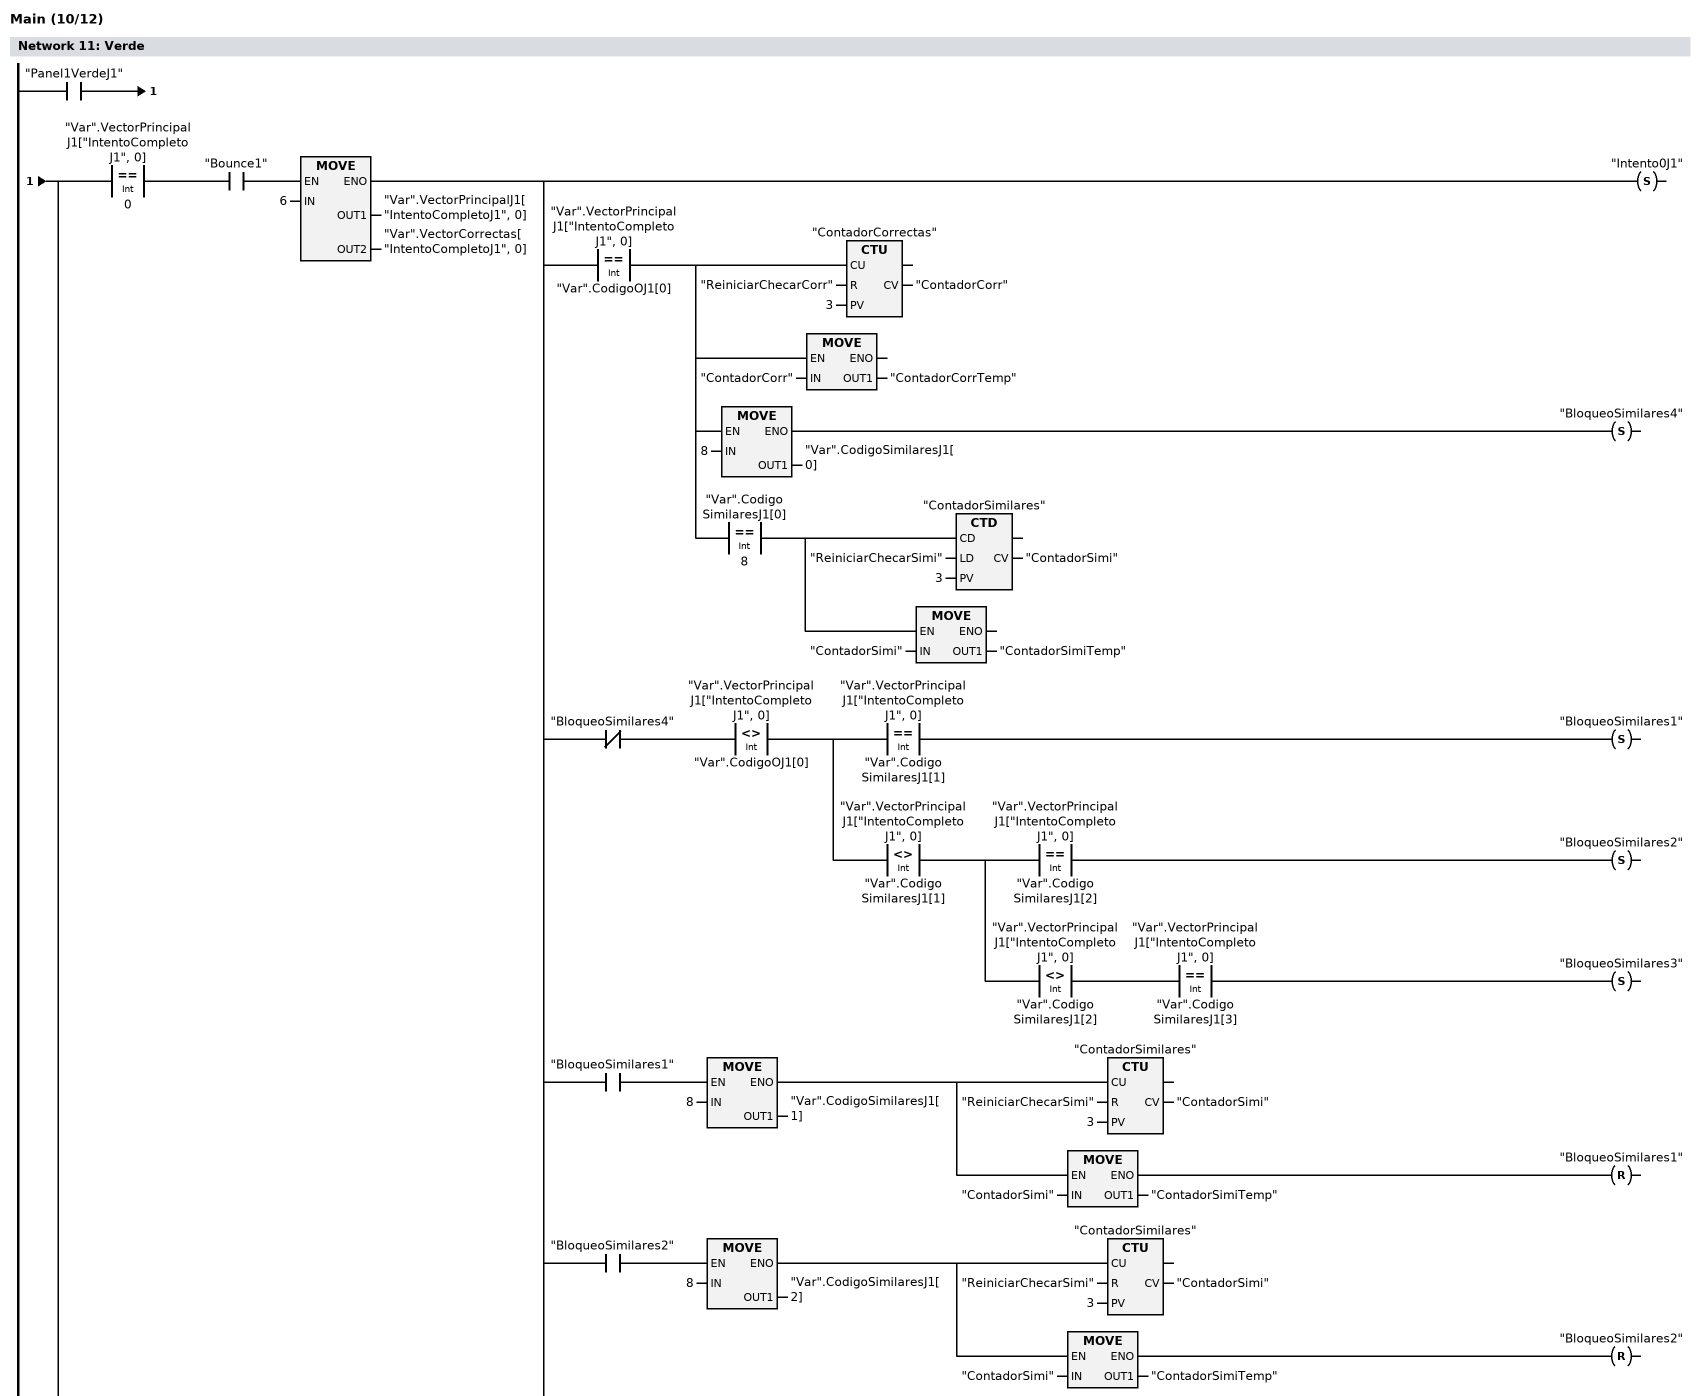
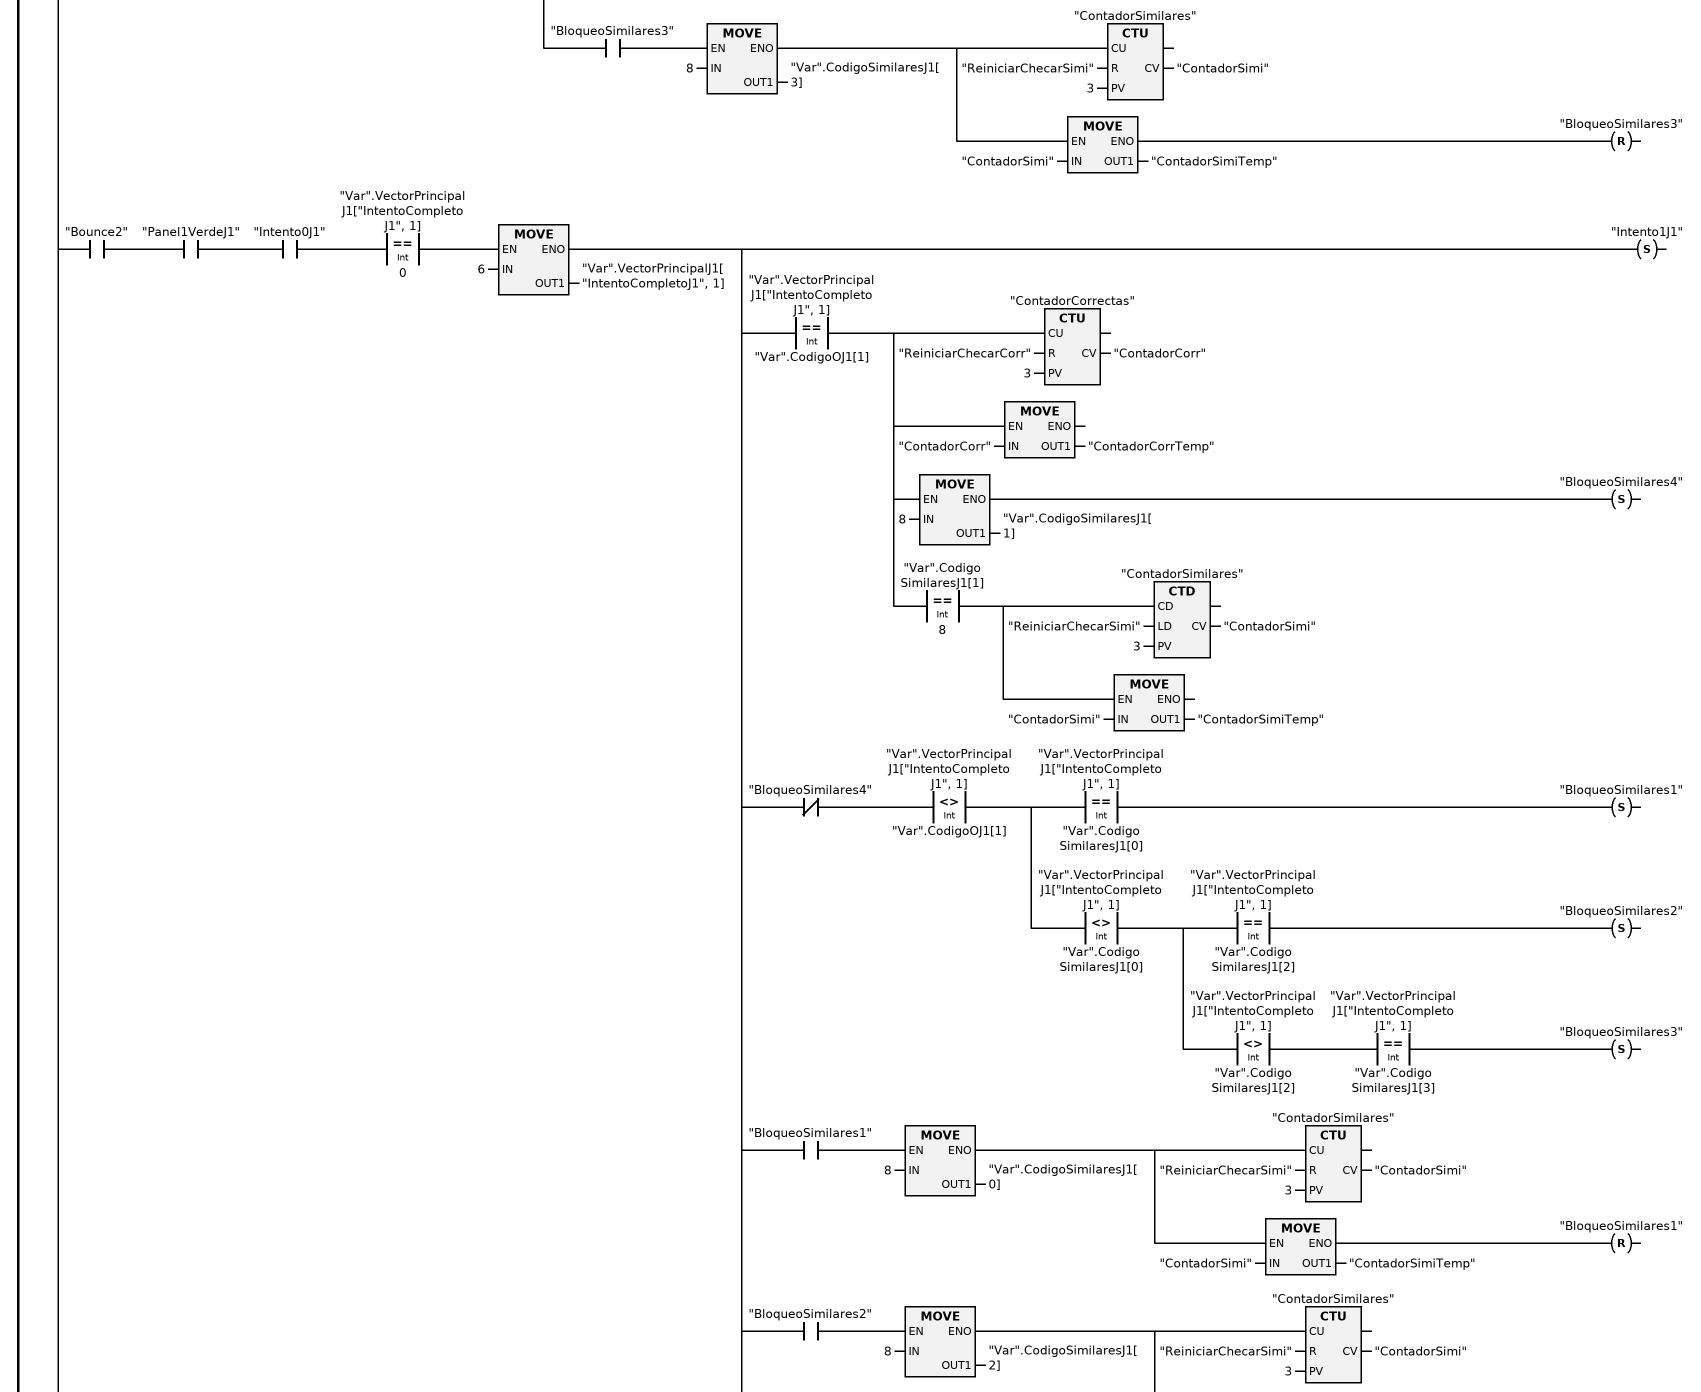
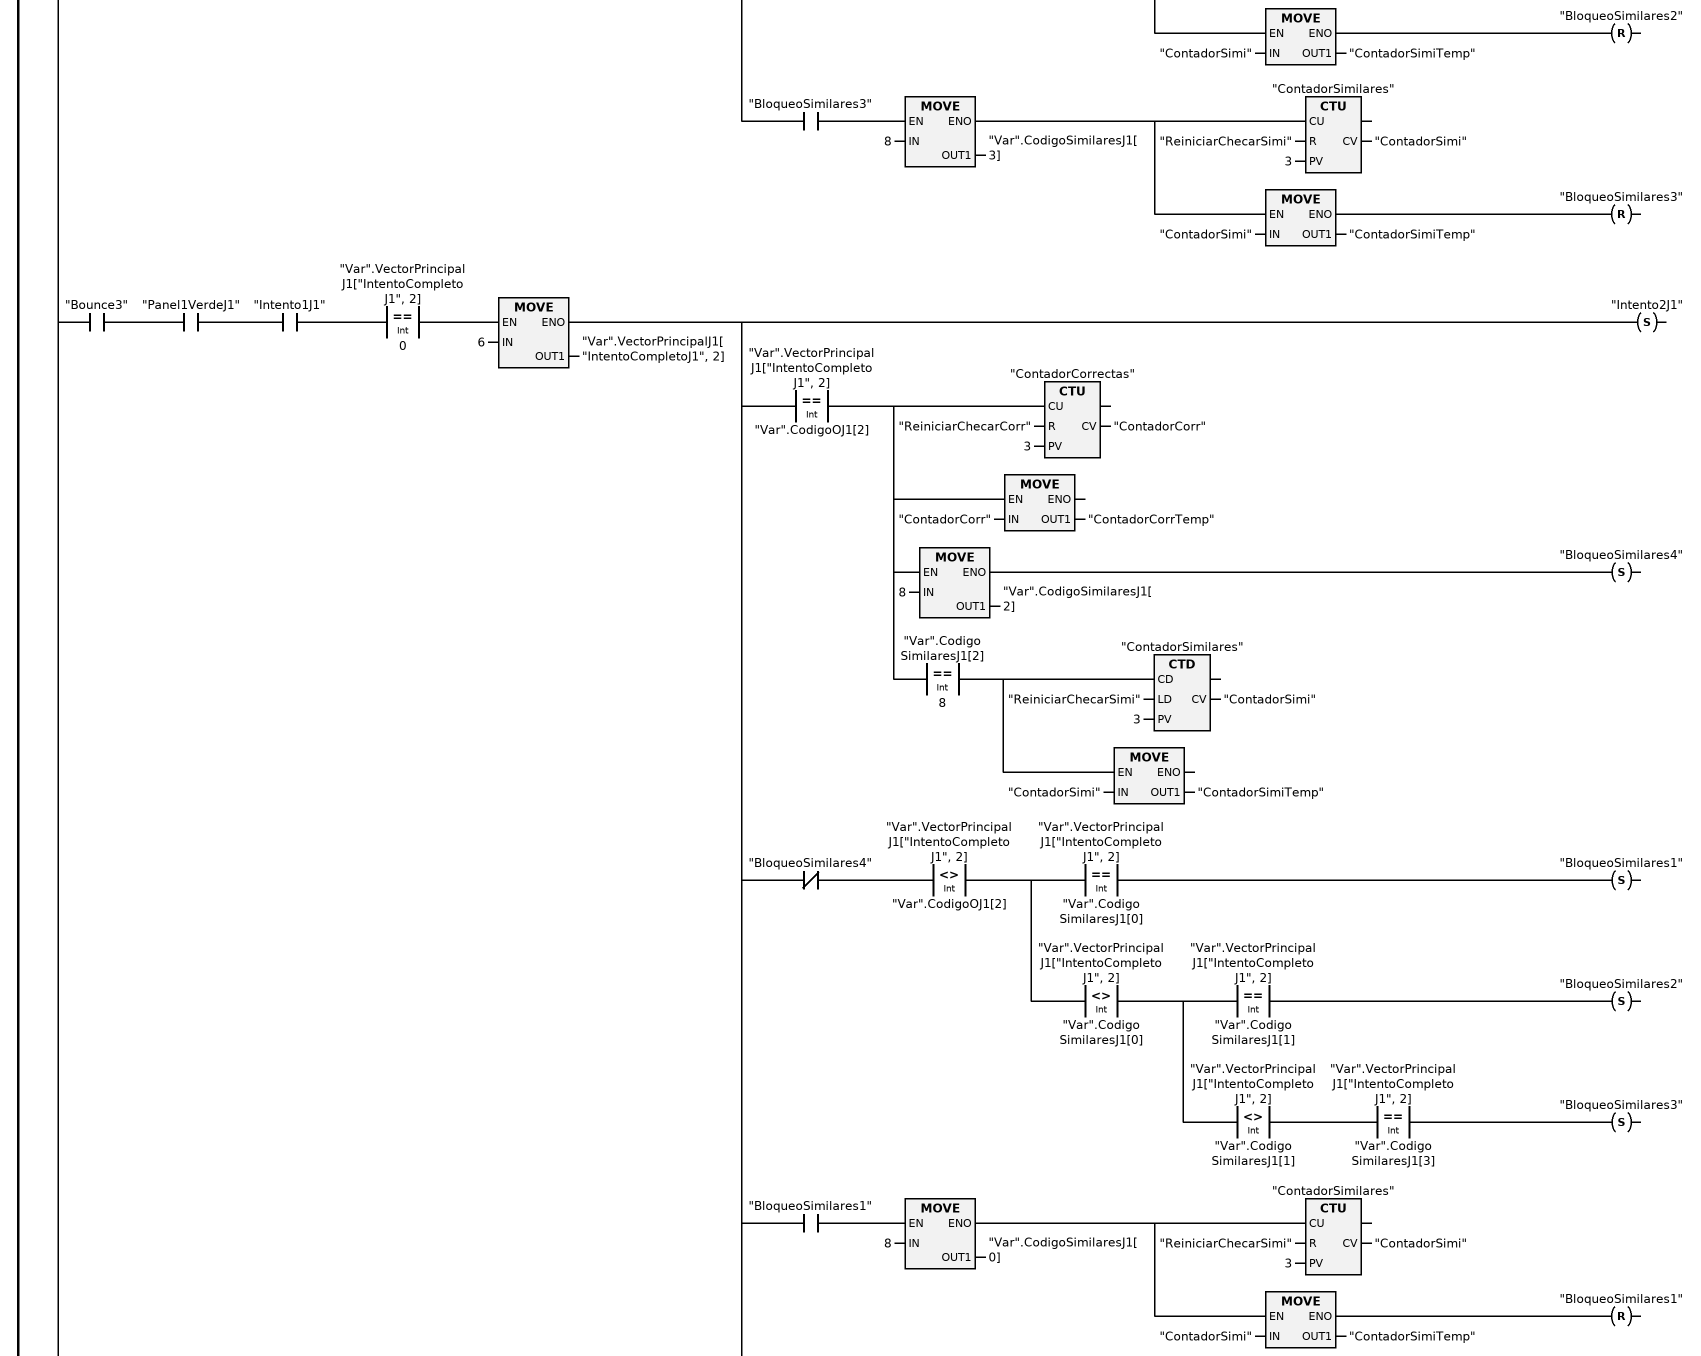
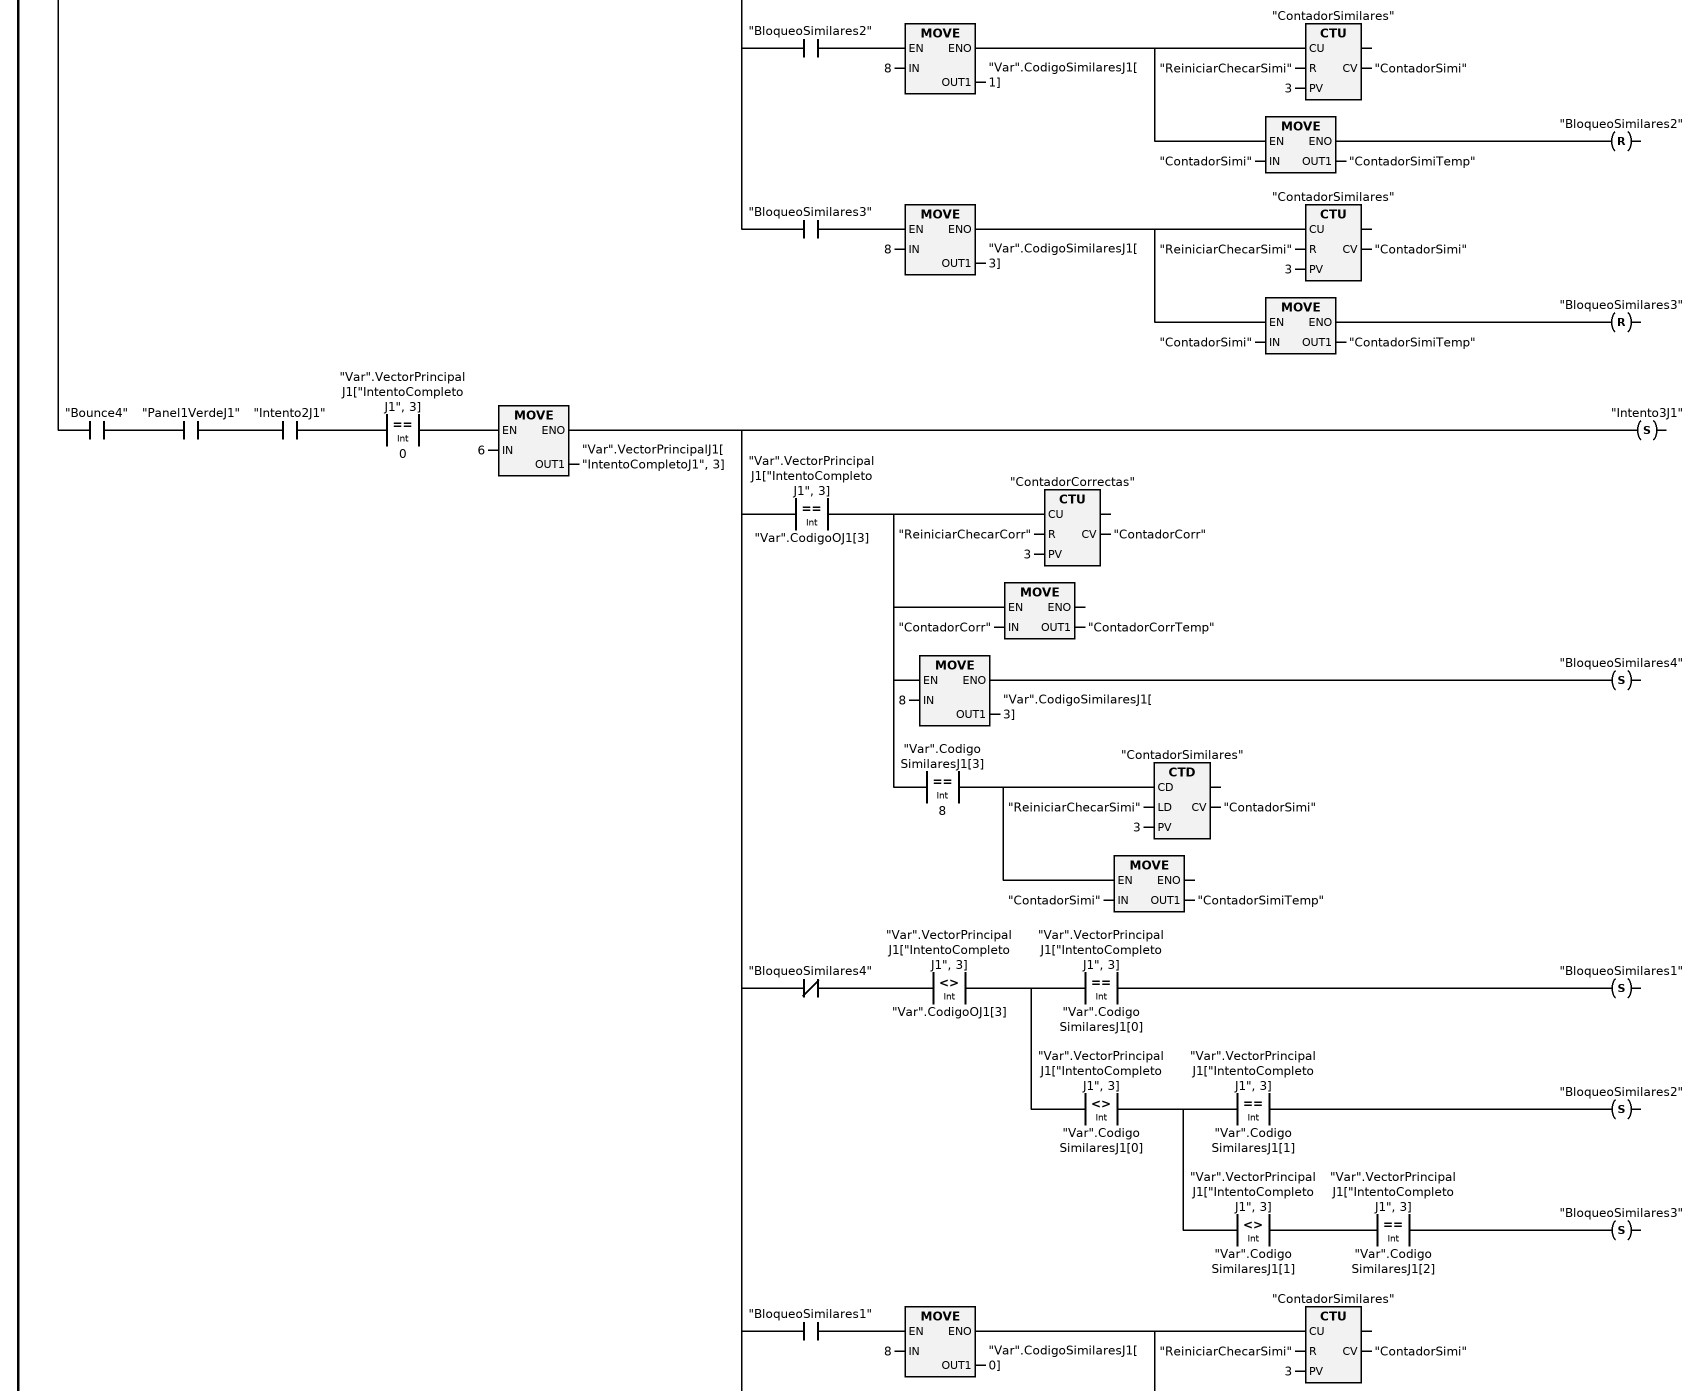
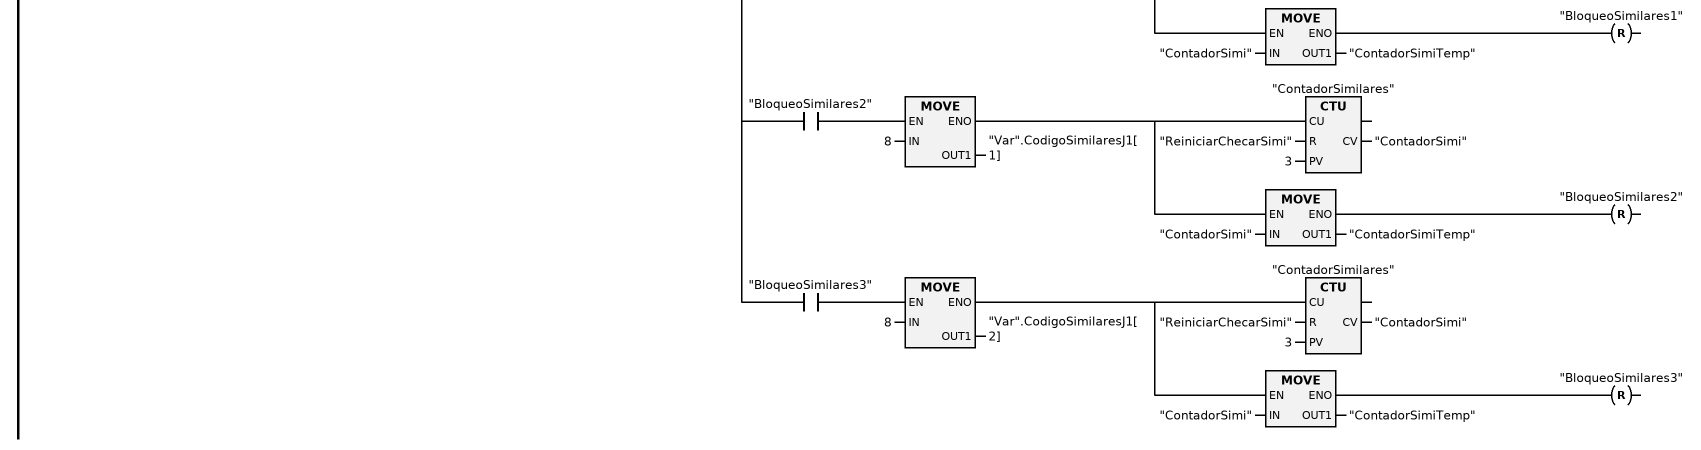
   #_w1 := "Panel1VerdeJ1" AND ("Var".VectorPrincipalJ1["IntentoCompletoJ1", 0] = 0) AND "Bounce1";
   IF #_w1 THEN
       "Var".VectorPrincipalJ1["IntentoCompletoJ1", 0] := 6;
       "Var".VectorCorrectas["IntentoCompletoJ1", 0] := 6;
       "Intento0J1" := TRUE;
   END_IF;
   #_w2 := #_w1 AND ("Var".VectorPrincipalJ1["IntentoCompletoJ1", 0] = "Var".CodigoOJ1[0]);
   "ContadorCorrectas".CTU(CU := #_w2, R := "ReiniciarChecarCorr", PV := 3, CV => "ContadorCorr");
   IF #_w2 THEN
       "ContadorCorrTemp" := "ContadorCorr";
       "Var".CodigoSimilaresJ1[0] := 8;
       "BloqueoSimilares4" := TRUE;
   END_IF;
   #_w3 := #_w2 AND ("Var".CodigoSimilaresJ1[0] = 8);
   "ContadorSimilares".CTD(CD := #_w3, LD := "ReiniciarChecarSimi", PV := 3, CV => "ContadorSimi");
   IF #_w3 THEN "ContadorSimiTemp" := "ContadorSimi"; END_IF;
   #_w4 := #_w1 AND NOT "BloqueoSimilares4" AND ("Var".VectorPrincipalJ1["IntentoCompletoJ1", 0] <> "Var".CodigoOJ1[0]);
   IF #_w4 AND ("Var".VectorPrincipalJ1["IntentoCompletoJ1", 0] = "Var".CodigoSimilaresJ1[1]) THEN
       "BloqueoSimilares1" := TRUE;
   END_IF;
   #_w5 := #_w4 AND ("Var".VectorPrincipalJ1["IntentoCompletoJ1", 0] <> "Var".CodigoSimilaresJ1[1]);
   IF #_w5 AND ("Var".VectorPrincipalJ1["IntentoCompletoJ1", 0] = "Var".CodigoSimilaresJ1[2]) THEN
       "BloqueoSimilares2" := TRUE;
   END_IF;
   IF #_w5 AND ("Var".VectorPrincipalJ1["IntentoCompletoJ1", 0] <> "Var".CodigoSimilaresJ1[2]) AND ("Var".VectorPrincipalJ1["IntentoCompletoJ1", 0] = "Var".CodigoSimilaresJ1[3]) THEN
       "BloqueoSimilares3" := TRUE;
   END_IF;
   #_w6 := #_w1 AND "BloqueoSimilares1";
   IF #_w6 THEN "Var".CodigoSimilaresJ1[1] := 8; END_IF;
   "ContadorSimilares".CTU(CU := #_w6, R := "ReiniciarChecarSimi", PV := 3, CV => "ContadorSimi");
   IF #_w6 THEN
       "ContadorSimiTemp" := "ContadorSimi";
       "BloqueoSimilares1" := FALSE;
   END_IF;
   #_w7 := #_w1 AND "BloqueoSimilares2";
   IF #_w7 THEN "Var".CodigoSimilaresJ1[2] := 8; END_IF;
   "ContadorSimilares".CTU(CU := #_w7, R := "ReiniciarChecarSimi", PV := 3, CV => "ContadorSimi");
   IF #_w7 THEN
       "ContadorSimiTemp" := "ContadorSimi";
       "BloqueoSimilares2" := FALSE;
   END_IF;
   #_w8 := #_w1 AND "BloqueoSimilares3";
   IF #_w8 THEN "Var".CodigoSimilaresJ1[3] := 8; END_IF;
   "ContadorSimilares".CTU(CU := #_w8, R := "ReiniciarChecarSimi", PV := 3, CV => "ContadorSimi");
   IF #_w8 THEN
       "ContadorSimiTemp" := "ContadorSimi";
       "BloqueoSimilares3" := FALSE;
   END_IF;
   #_w9 := "Panel1VerdeJ1" AND "Bounce2" AND "Panel1VerdeJ1" AND "Intento0J1" AND ("Var".VectorPrincipalJ1["IntentoCompletoJ1", 1] = 0);
   IF #_w9 THEN
       "Var".VectorPrincipalJ1["IntentoCompletoJ1", 1] := 6;
       "Intento1J1" := TRUE;
   END_IF;
   #_w10 := #_w9 AND ("Var".VectorPrincipalJ1["IntentoCompletoJ1", 1] = "Var".CodigoOJ1[1]);
   "ContadorCorrectas".CTU(CU := #_w10, R := "ReiniciarChecarCorr", PV := 3, CV => "ContadorCorr");
   IF #_w10 THEN
       "ContadorCorrTemp" := "ContadorCorr";
       "Var".CodigoSimilaresJ1[1] := 8;
       "BloqueoSimilares4" := TRUE;
   END_IF;
   #_w11 := #_w10 AND ("Var".CodigoSimilaresJ1[1] = 8);
   "ContadorSimilares".CTD(CD := #_w11, LD := "ReiniciarChecarSimi", PV := 3, CV => "ContadorSimi");
   IF #_w11 THEN "ContadorSimiTemp" := "ContadorSimi"; END_IF;
   #_w12 := #_w9 AND NOT "BloqueoSimilares4" AND ("Var".VectorPrincipalJ1["IntentoCompletoJ1", 1] <> "Var".CodigoOJ1[1]);
   IF #_w12 AND ("Var".VectorPrincipalJ1["IntentoCompletoJ1", 1] = "Var".CodigoSimilaresJ1[0]) THEN
       "BloqueoSimilares1" := TRUE;
   END_IF;
   #_w13 := #_w12 AND ("Var".VectorPrincipalJ1["IntentoCompletoJ1", 1] <> "Var".CodigoSimilaresJ1[0]);
   IF #_w13 AND ("Var".VectorPrincipalJ1["IntentoCompletoJ1", 1] = "Var".CodigoSimilaresJ1[2]) THEN
       "BloqueoSimilares2" := TRUE;
   END_IF;
   IF #_w13 AND ("Var".VectorPrincipalJ1["IntentoCompletoJ1", 1] <> "Var".CodigoSimilaresJ1[2]) AND ("Var".VectorPrincipalJ1["IntentoCompletoJ1", 1] = "Var".CodigoSimilaresJ1[3]) THEN
       "BloqueoSimilares3" := TRUE;
   END_IF;
   #_w14 := #_w9 AND "BloqueoSimilares1";
   IF #_w14 THEN "Var".CodigoSimilaresJ1[0] := 8; END_IF;
   "ContadorSimilares".CTU(CU := #_w14, R := "ReiniciarChecarSimi", PV := 3, CV => "ContadorSimi");
   IF #_w14 THEN
       "ContadorSimiTemp" := "ContadorSimi";
       "BloqueoSimilares1" := FALSE;
   END_IF;
   #_w15 := #_w9 AND "BloqueoSimilares2";
   IF #_w15 THEN "Var".CodigoSimilaresJ1[2] := 8; END_IF;
   "ContadorSimilares".CTU(CU := #_w15, R := "ReiniciarChecarSimi", PV := 3, CV => "ContadorSimi");
   IF #_w15 THEN
       "ContadorSimiTemp" := "ContadorSimi";
       "BloqueoSimilares2" := FALSE;
   END_IF;
   #_w16 := #_w9 AND "BloqueoSimilares3";
   IF #_w16 THEN "Var".CodigoSimilaresJ1[3] := 8; END_IF;
   "ContadorSimilares".CTU(CU := #_w16, R := "ReiniciarChecarSimi", PV := 3, CV => "ContadorSimi");
   IF #_w16 THEN
       "ContadorSimiTemp" := "ContadorSimi";
       "BloqueoSimilares3" := FALSE;
   END_IF;
   #_w17 := "Panel1VerdeJ1" AND "Bounce3" AND "Panel1VerdeJ1" AND "Intento1J1" AND ("Var".VectorPrincipalJ1["IntentoCompletoJ1", 2] = 0);
   IF #_w17 THEN
       "Var".VectorPrincipalJ1["IntentoCompletoJ1", 2] := 6;
       "Intento2J1" := TRUE;
   END_IF;
   #_w18 := #_w17 AND ("Var".VectorPrincipalJ1["IntentoCompletoJ1", 2] = "Var".CodigoOJ1[2]);
   "ContadorCorrectas".CTU(CU := #_w18, R := "ReiniciarChecarCorr", PV := 3, CV => "ContadorCorr");
   IF #_w18 THEN
       "ContadorCorrTemp" := "ContadorCorr";
       "Var".CodigoSimilaresJ1[2] := 8;
       "BloqueoSimilares4" := TRUE;
   END_IF;
   #_w19 := #_w18 AND ("Var".CodigoSimilaresJ1[2] = 8);
   "ContadorSimilares".CTD(CD := #_w19, LD := "ReiniciarChecarSimi", PV := 3, CV => "ContadorSimi");
   IF #_w19 THEN "ContadorSimiTemp" := "ContadorSimi"; END_IF;
   #_w20 := #_w17 AND NOT "BloqueoSimilares4" AND ("Var".VectorPrincipalJ1["IntentoCompletoJ1", 2] <> "Var".CodigoOJ1[2]);
   IF #_w20 AND ("Var".VectorPrincipalJ1["IntentoCompletoJ1", 2] = "Var".CodigoSimilaresJ1[0]) THEN
       "BloqueoSimilares1" := TRUE;
   END_IF;
   #_w21 := #_w20 AND ("Var".VectorPrincipalJ1["IntentoCompletoJ1", 2] <> "Var".CodigoSimilaresJ1[0]);
   IF #_w21 AND ("Var".VectorPrincipalJ1["IntentoCompletoJ1", 2] = "Var".CodigoSimilaresJ1[1]) THEN
       "BloqueoSimilares2" := TRUE;
   END_IF;
   IF #_w21 AND ("Var".VectorPrincipalJ1["IntentoCompletoJ1", 2] <> "Var".CodigoSimilaresJ1[1]) AND ("Var".VectorPrincipalJ1["IntentoCompletoJ1", 2] = "Var".CodigoSimilaresJ1[3]) THEN
       "BloqueoSimilares3" := TRUE;
   END_IF;
   #_w22 := #_w17 AND "BloqueoSimilares1";
   IF #_w22 THEN "Var".CodigoSimilaresJ1[0] := 8; END_IF;
   "ContadorSimilares".CTU(CU := #_w22, R := "ReiniciarChecarSimi", PV := 3, CV => "ContadorSimi");
   IF #_w22 THEN
       "ContadorSimiTemp" := "ContadorSimi";
       "BloqueoSimilares1" := FALSE;
   END_IF;
   #_w23 := #_w17 AND "BloqueoSimilares2";
   IF #_w23 THEN "Var".CodigoSimilaresJ1[1] := 8; END_IF;
   "ContadorSimilares".CTU(CU := #_w23, R := "ReiniciarChecarSimi", PV := 3, CV => "ContadorSimi");
   IF #_w23 THEN
       "ContadorSimiTemp" := "ContadorSimi";
       "BloqueoSimilares2" := FALSE;
   END_IF;
   #_w24 := #_w17 AND "BloqueoSimilares3";
   IF #_w24 THEN "Var".CodigoSimilaresJ1[3] := 8; END_IF;
   "ContadorSimilares".CTU(CU := #_w24, R := "ReiniciarChecarSimi", PV := 3, CV => "ContadorSimi");
   IF #_w24 THEN
       "ContadorSimiTemp" := "ContadorSimi";
       "BloqueoSimilares3" := FALSE;
   END_IF;
   #_w25 := "Panel1VerdeJ1" AND "Bounce4" AND "Panel1VerdeJ1" AND "Intento2J1" AND ("Var".VectorPrincipalJ1["IntentoCompletoJ1", 3] = 0);
   IF #_w25 THEN
       "Var".VectorPrincipalJ1["IntentoCompletoJ1", 3] := 6;
       "Intento3J1" := TRUE;
   END_IF;
   #_w26 := #_w25 AND ("Var".VectorPrincipalJ1["IntentoCompletoJ1", 3] = "Var".CodigoOJ1[3]);
   "ContadorCorrectas".CTU(CU := #_w26, R := "ReiniciarChecarCorr", PV := 3, CV => "ContadorCorr");
   IF #_w26 THEN
       "ContadorCorrTemp" := "ContadorCorr";
       "Var".CodigoSimilaresJ1[3] := 8;
       "BloqueoSimilares4" := TRUE;
   END_IF;
   #_w27 := #_w26 AND ("Var".CodigoSimilaresJ1[3] = 8);
   "ContadorSimilares".CTD(CD := #_w27, LD := "ReiniciarChecarSimi", PV := 3, CV => "ContadorSimi");
   IF #_w27 THEN "ContadorSimiTemp" := "ContadorSimi"; END_IF;
   #_w28 := #_w25 AND NOT "BloqueoSimilares4" AND ("Var".VectorPrincipalJ1["IntentoCompletoJ1", 3] <> "Var".CodigoOJ1[3]);
   IF #_w28 AND ("Var".VectorPrincipalJ1["IntentoCompletoJ1", 3] = "Var".CodigoSimilaresJ1[0]) THEN
       "BloqueoSimilares1" := TRUE;
   END_IF;
   #_w29 := #_w28 AND ("Var".VectorPrincipalJ1["IntentoCompletoJ1", 3] <> "Var".CodigoSimilaresJ1[0]);
   IF #_w29 AND ("Var".VectorPrincipalJ1["IntentoCompletoJ1", 3] = "Var".CodigoSimilaresJ1[1]) THEN
       "BloqueoSimilares2" := TRUE;
   END_IF;
   IF #_w29 AND ("Var".VectorPrincipalJ1["IntentoCompletoJ1", 3] <> "Var".CodigoSimilaresJ1[1]) AND ("Var".VectorPrincipalJ1["IntentoCompletoJ1", 3] = "Var".CodigoSimilaresJ1[2]) THEN
       "BloqueoSimilares3" := TRUE;
   END_IF;
   #_w30 := #_w25 AND "BloqueoSimilares1";
   IF #_w30 THEN "Var".CodigoSimilaresJ1[0] := 8; END_IF;
   "ContadorSimilares".CTU(CU := #_w30, R := "ReiniciarChecarSimi", PV := 3, CV => "ContadorSimi");
   IF #_w30 THEN
       "ContadorSimiTemp" := "ContadorSimi";
       "BloqueoSimilares1" := FALSE;
   END_IF;
   #_w31 := #_w25 AND "BloqueoSimilares2";
   IF #_w31 THEN "Var".CodigoSimilaresJ1[1] := 8; END_IF;
   "ContadorSimilares".CTU(CU := #_w31, R := "ReiniciarChecarSimi", PV := 3, CV => "ContadorSimi");
   IF #_w31 THEN
       "ContadorSimiTemp" := "ContadorSimi";
       "BloqueoSimilares2" := FALSE;
   END_IF;
   #_w32 := #_w25 AND "BloqueoSimilares3";
   IF #_w32 THEN "Var".CodigoSimilaresJ1[2] := 8; END_IF;
   "ContadorSimilares".CTU(CU := #_w32, R := "ReiniciarChecarSimi", PV := 3, CV => "ContadorSimi");
   IF #_w32 THEN
       "ContadorSimiTemp" := "ContadorSimi";
       "BloqueoSimilares3" := FALSE;
   END_IF;
END_REGION

REGION Network 12: Amarillo
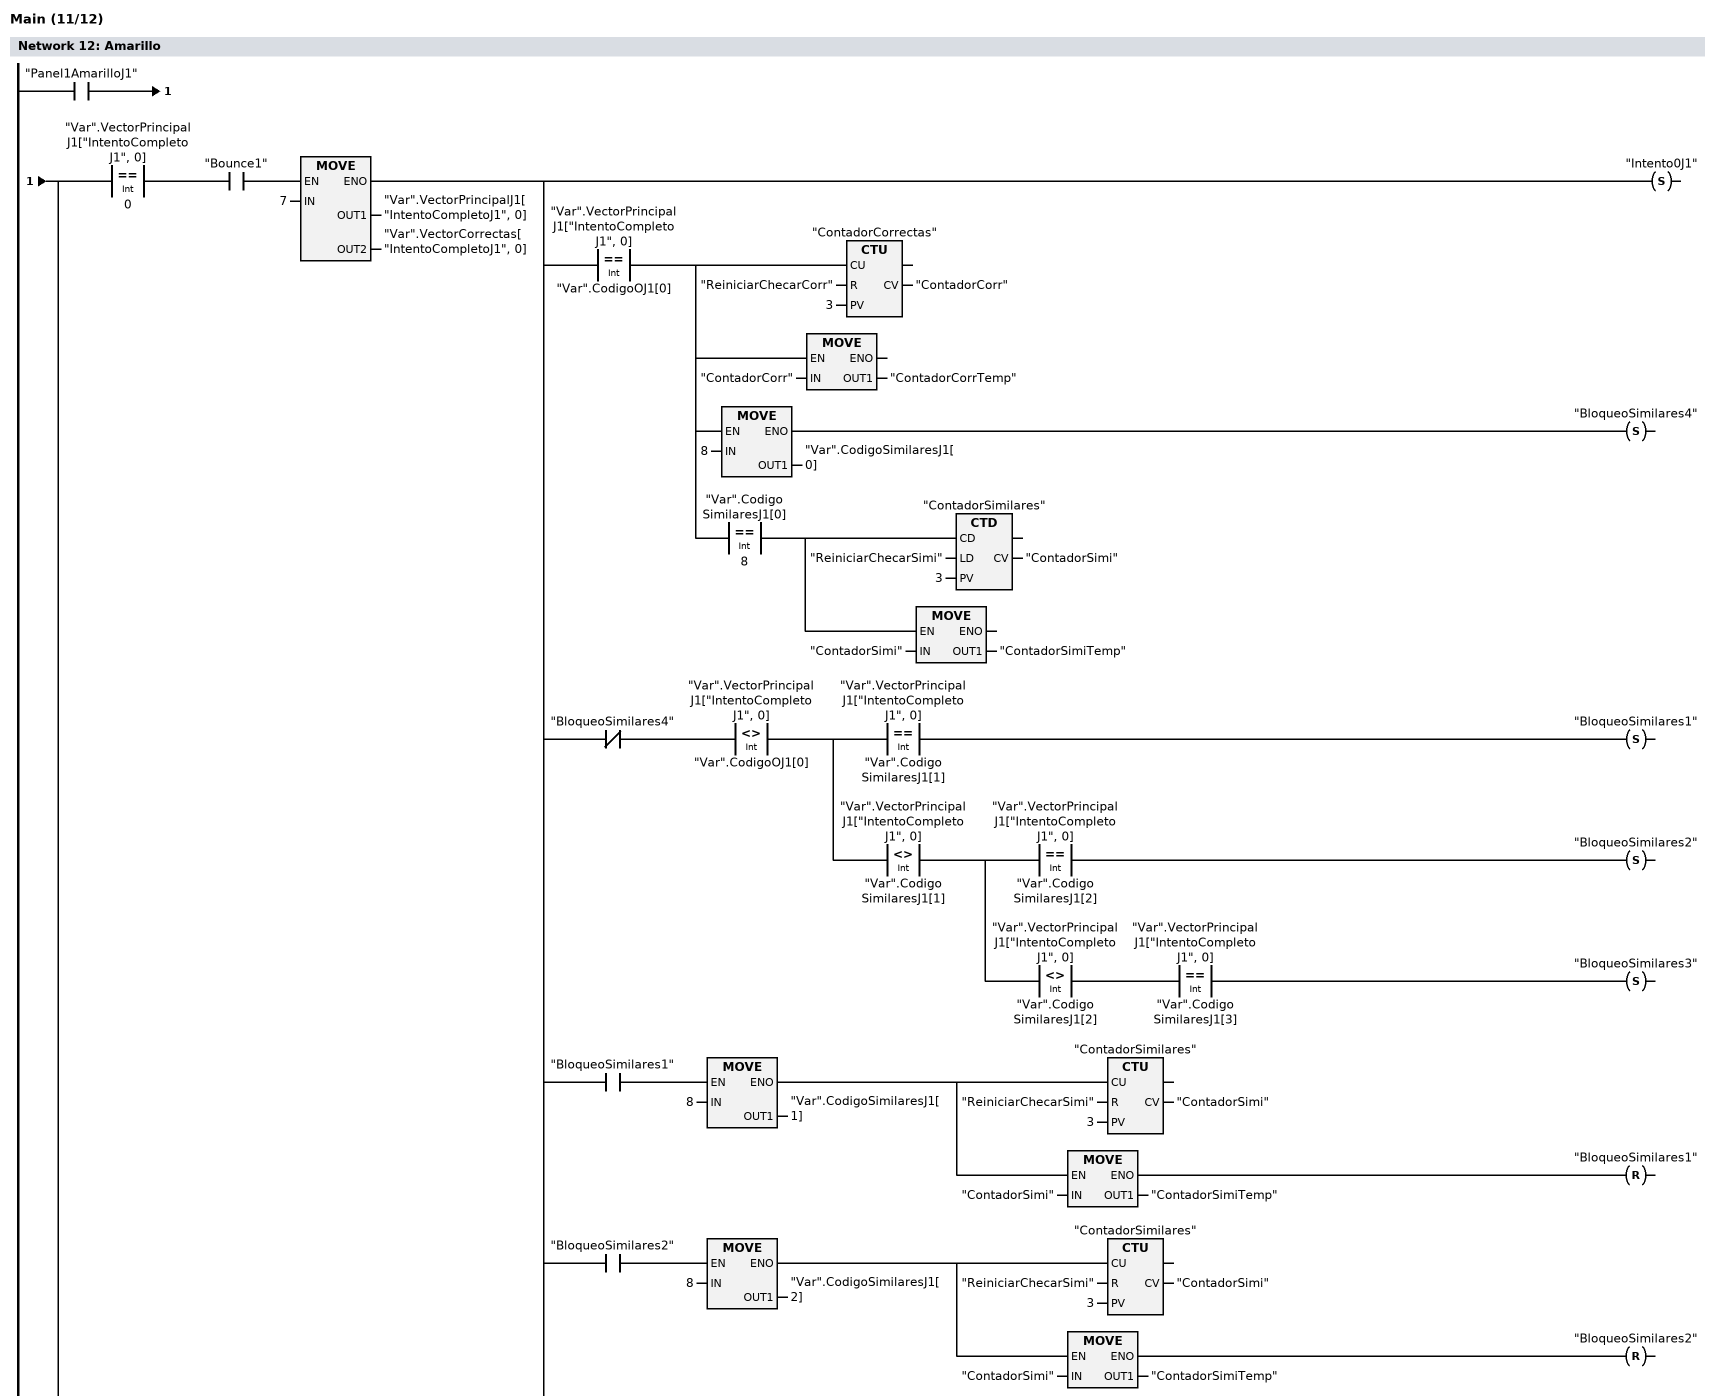
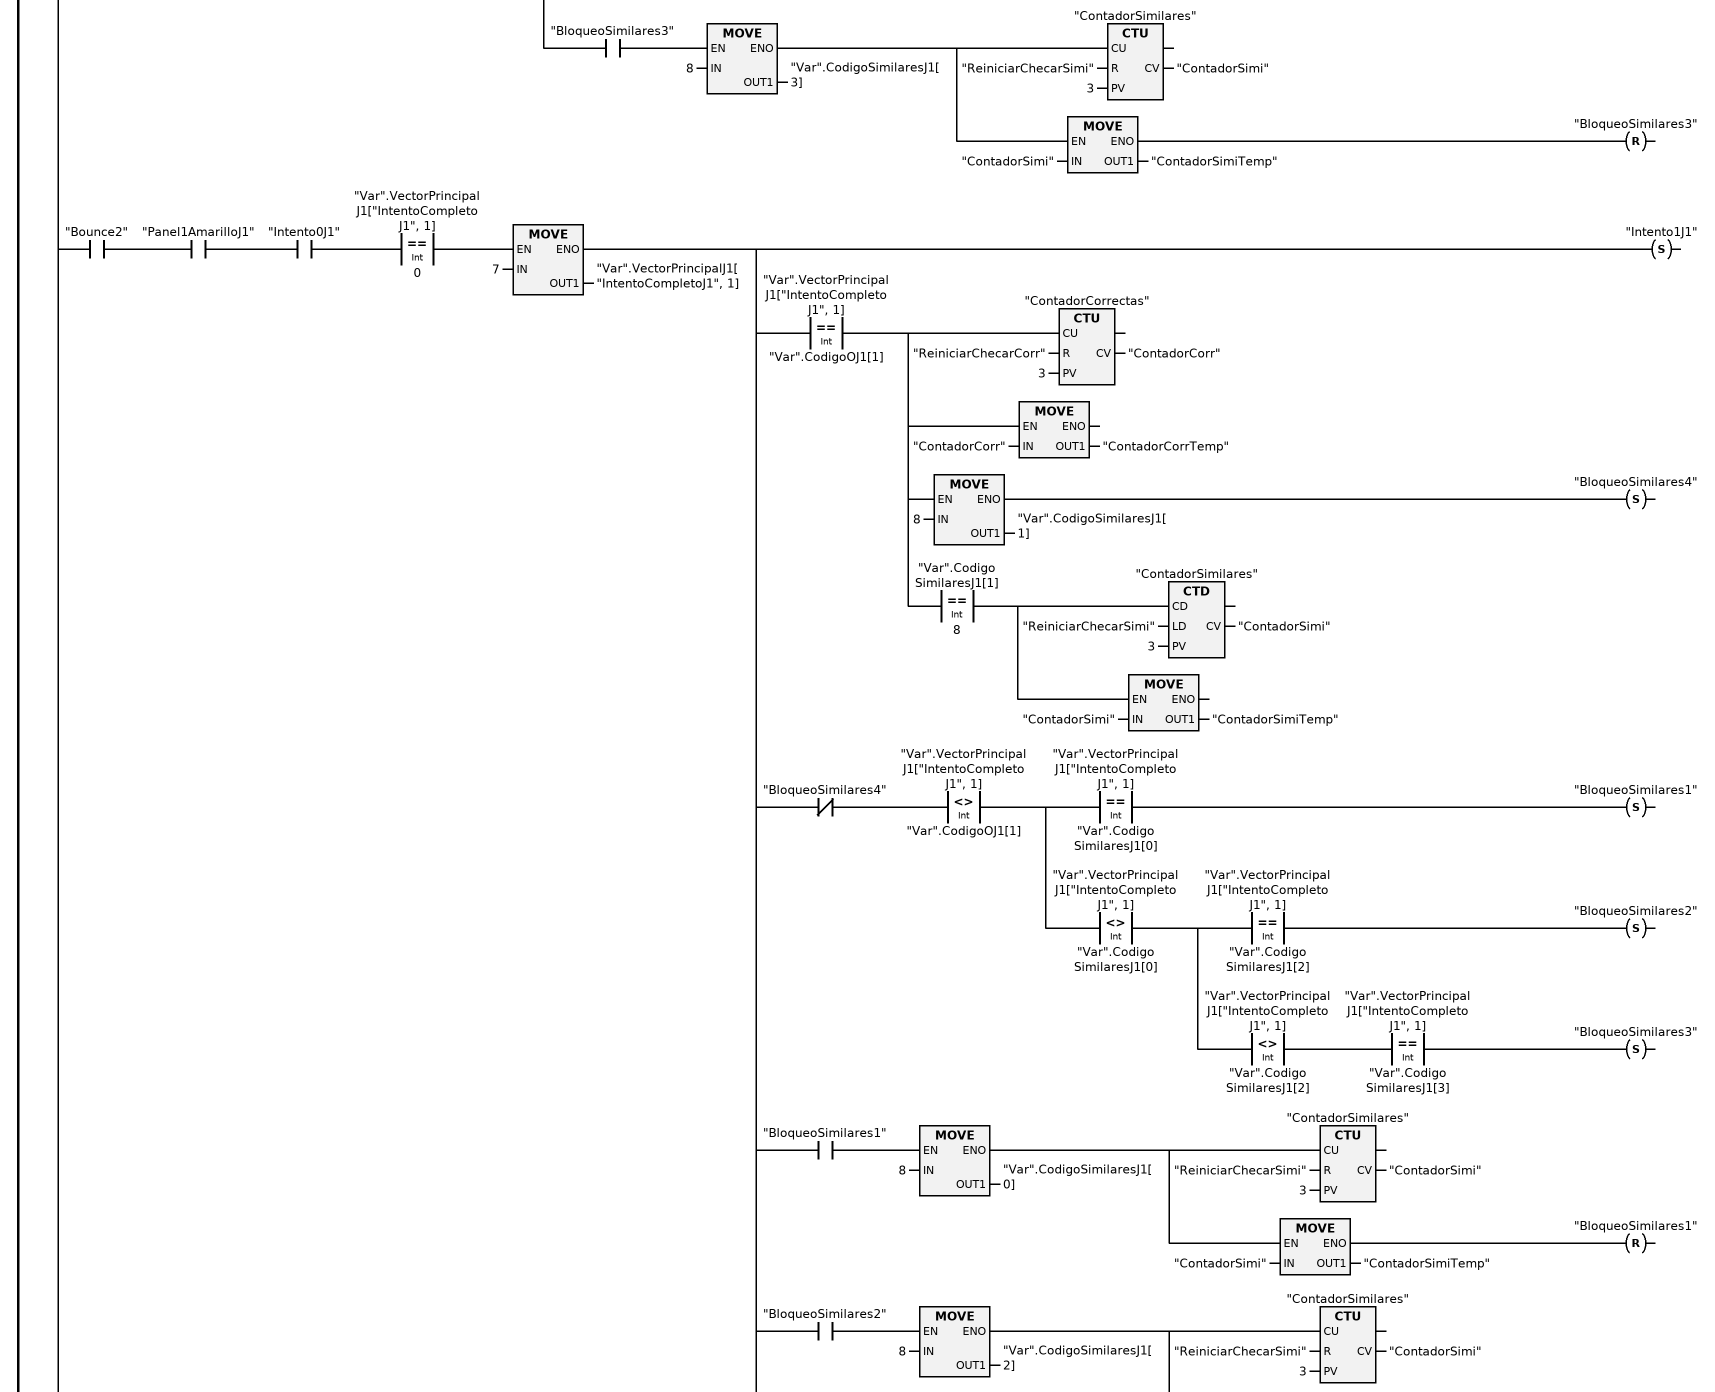
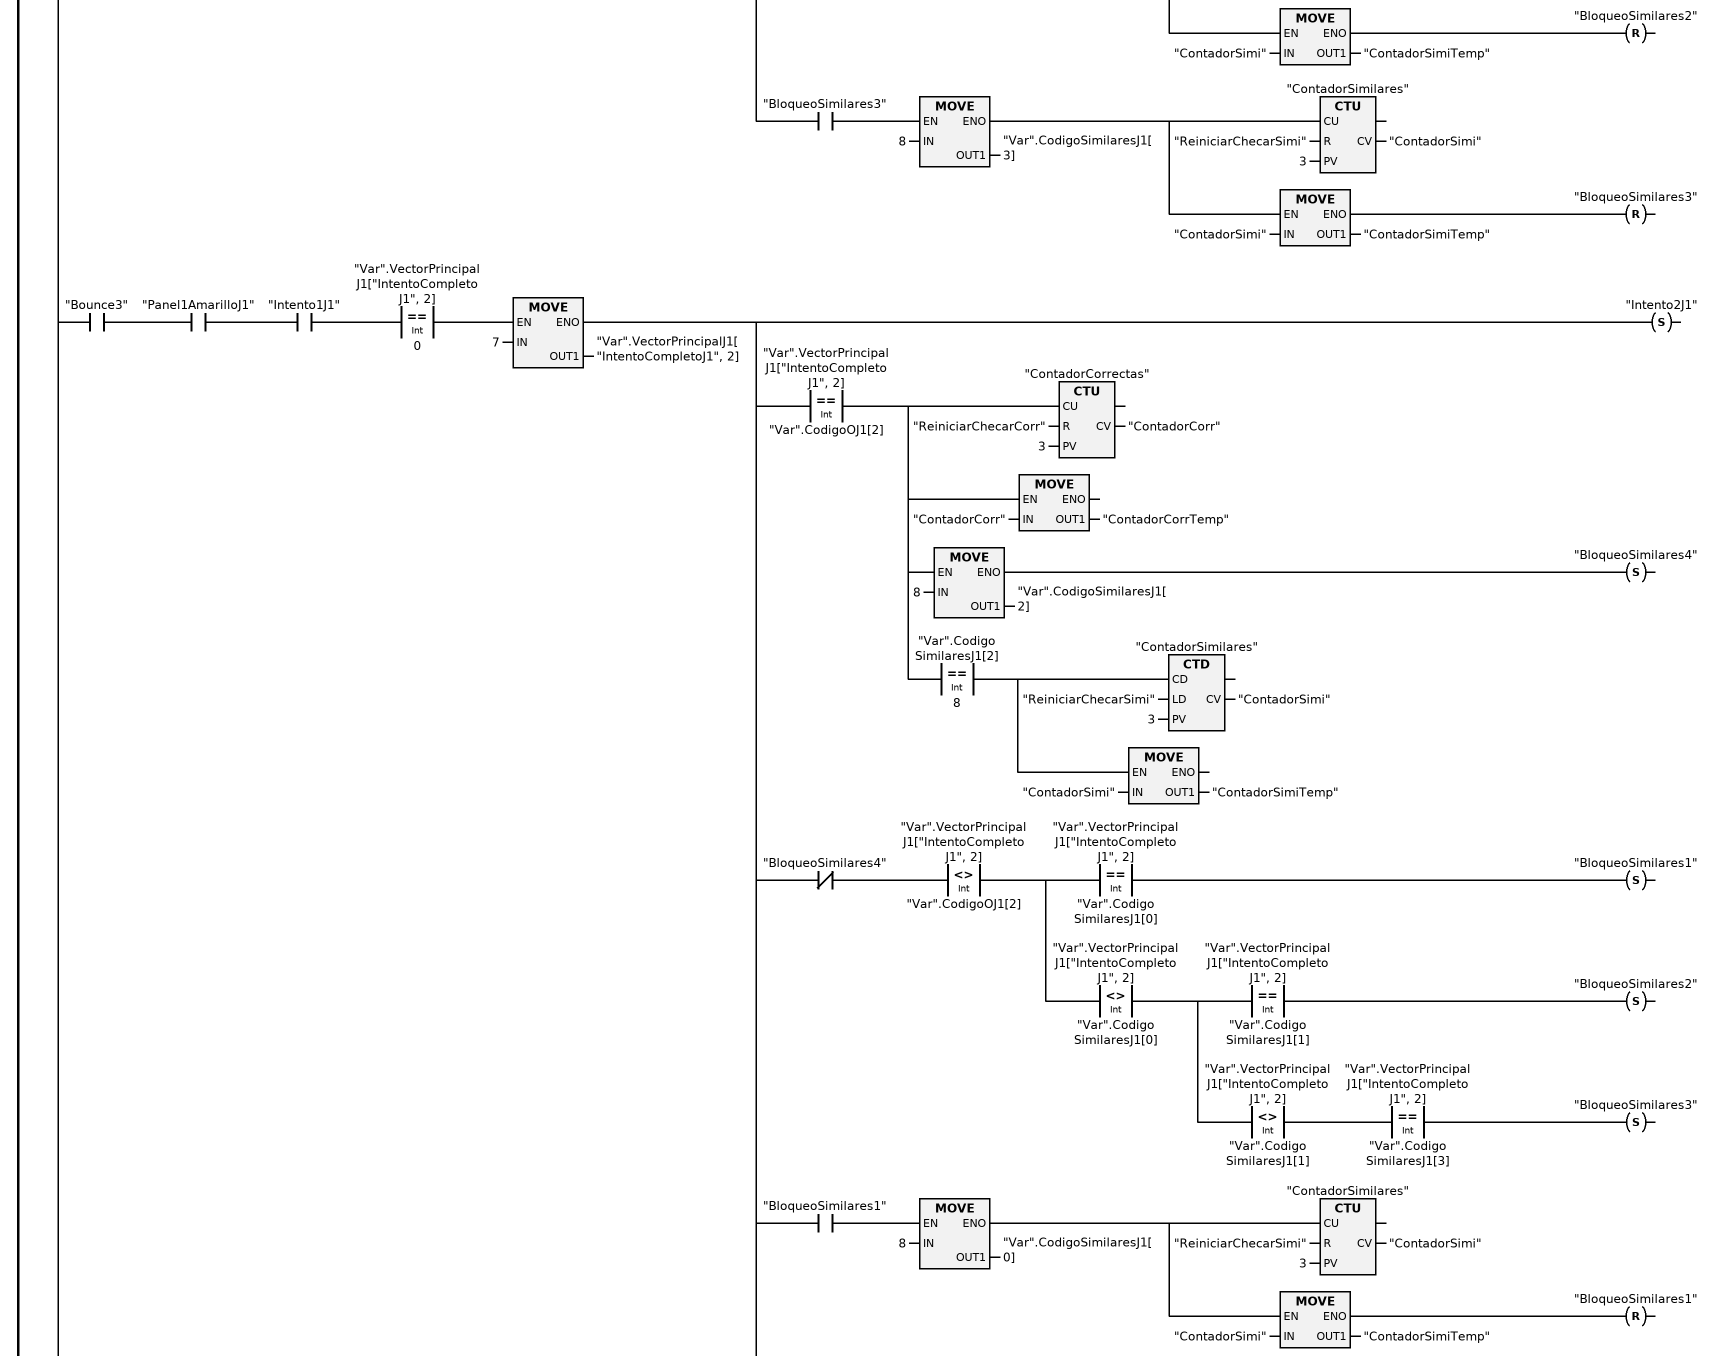
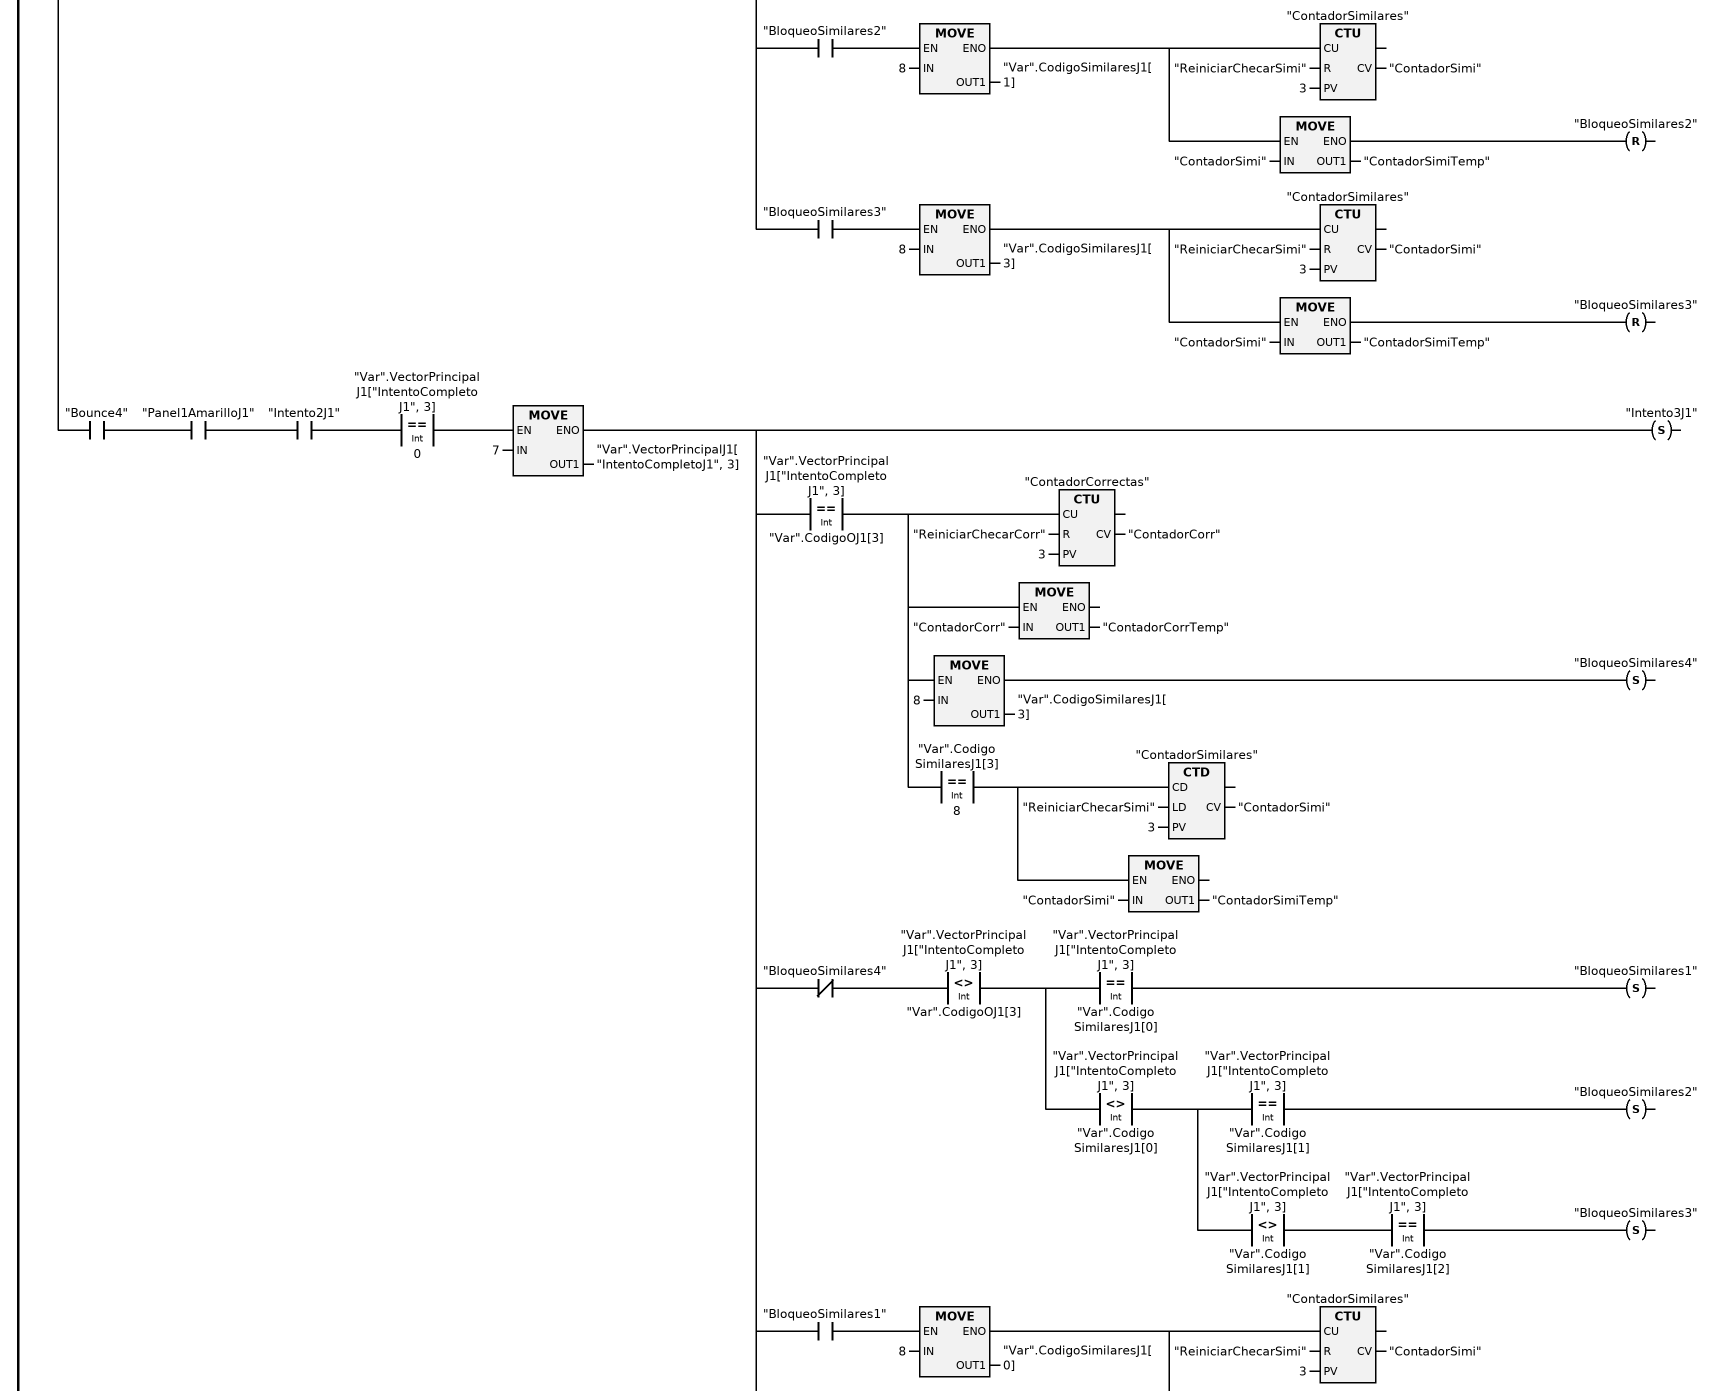
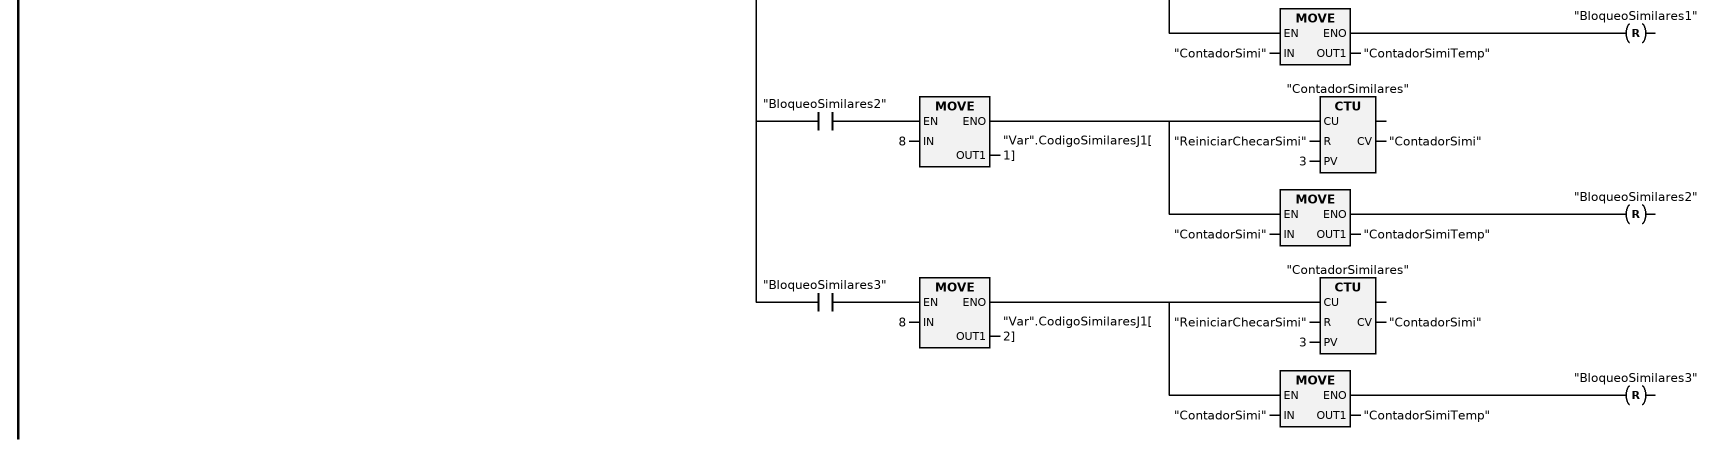
   #_w1 := "Panel1AmarilloJ1" AND ("Var".VectorPrincipalJ1["IntentoCompletoJ1", 0] = 0) AND "Bounce1";
   IF #_w1 THEN
       "Var".VectorPrincipalJ1["IntentoCompletoJ1", 0] := 7;
       "Var".VectorCorrectas["IntentoCompletoJ1", 0] := 7;
       "Intento0J1" := TRUE;
   END_IF;
   #_w2 := #_w1 AND ("Var".VectorPrincipalJ1["IntentoCompletoJ1", 0] = "Var".CodigoOJ1[0]);
   "ContadorCorrectas".CTU(CU := #_w2, R := "ReiniciarChecarCorr", PV := 3, CV => "ContadorCorr");
   IF #_w2 THEN
       "ContadorCorrTemp" := "ContadorCorr";
       "Var".CodigoSimilaresJ1[0] := 8;
       "BloqueoSimilares4" := TRUE;
   END_IF;
   #_w3 := #_w2 AND ("Var".CodigoSimilaresJ1[0] = 8);
   "ContadorSimilares".CTD(CD := #_w3, LD := "ReiniciarChecarSimi", PV := 3, CV => "ContadorSimi");
   IF #_w3 THEN "ContadorSimiTemp" := "ContadorSimi"; END_IF;
   #_w4 := #_w1 AND NOT "BloqueoSimilares4" AND ("Var".VectorPrincipalJ1["IntentoCompletoJ1", 0] <> "Var".CodigoOJ1[0]);
   IF #_w4 AND ("Var".VectorPrincipalJ1["IntentoCompletoJ1", 0] = "Var".CodigoSimilaresJ1[1]) THEN
       "BloqueoSimilares1" := TRUE;
   END_IF;
   #_w5 := #_w4 AND ("Var".VectorPrincipalJ1["IntentoCompletoJ1", 0] <> "Var".CodigoSimilaresJ1[1]);
   IF #_w5 AND ("Var".VectorPrincipalJ1["IntentoCompletoJ1", 0] = "Var".CodigoSimilaresJ1[2]) THEN
       "BloqueoSimilares2" := TRUE;
   END_IF;
   IF #_w5 AND ("Var".VectorPrincipalJ1["IntentoCompletoJ1", 0] <> "Var".CodigoSimilaresJ1[2]) AND ("Var".VectorPrincipalJ1["IntentoCompletoJ1", 0] = "Var".CodigoSimilaresJ1[3]) THEN
       "BloqueoSimilares3" := TRUE;
   END_IF;
   #_w6 := #_w1 AND "BloqueoSimilares1";
   IF #_w6 THEN "Var".CodigoSimilaresJ1[1] := 8; END_IF;
   "ContadorSimilares".CTU(CU := #_w6, R := "ReiniciarChecarSimi", PV := 3, CV => "ContadorSimi");
   IF #_w6 THEN
       "ContadorSimiTemp" := "ContadorSimi";
       "BloqueoSimilares1" := FALSE;
   END_IF;
   #_w7 := #_w1 AND "BloqueoSimilares2";
   IF #_w7 THEN "Var".CodigoSimilaresJ1[2] := 8; END_IF;
   "ContadorSimilares".CTU(CU := #_w7, R := "ReiniciarChecarSimi", PV := 3, CV => "ContadorSimi");
   IF #_w7 THEN
       "ContadorSimiTemp" := "ContadorSimi";
       "BloqueoSimilares2" := FALSE;
   END_IF;
   #_w8 := #_w1 AND "BloqueoSimilares3";
   IF #_w8 THEN "Var".CodigoSimilaresJ1[3] := 8; END_IF;
   "ContadorSimilares".CTU(CU := #_w8, R := "ReiniciarChecarSimi", PV := 3, CV => "ContadorSimi");
   IF #_w8 THEN
       "ContadorSimiTemp" := "ContadorSimi";
       "BloqueoSimilares3" := FALSE;
   END_IF;
   #_w9 := "Panel1AmarilloJ1" AND "Bounce2" AND "Panel1AmarilloJ1" AND "Intento0J1" AND ("Var".VectorPrincipalJ1["IntentoCompletoJ1", 1] = 0);
   IF #_w9 THEN
       "Var".VectorPrincipalJ1["IntentoCompletoJ1", 1] := 7;
       "Intento1J1" := TRUE;
   END_IF;
   #_w10 := #_w9 AND ("Var".VectorPrincipalJ1["IntentoCompletoJ1", 1] = "Var".CodigoOJ1[1]);
   "ContadorCorrectas".CTU(CU := #_w10, R := "ReiniciarChecarCorr", PV := 3, CV => "ContadorCorr");
   IF #_w10 THEN
       "ContadorCorrTemp" := "ContadorCorr";
       "Var".CodigoSimilaresJ1[1] := 8;
       "BloqueoSimilares4" := TRUE;
   END_IF;
   #_w11 := #_w10 AND ("Var".CodigoSimilaresJ1[1] = 8);
   "ContadorSimilares".CTD(CD := #_w11, LD := "ReiniciarChecarSimi", PV := 3, CV => "ContadorSimi");
   IF #_w11 THEN "ContadorSimiTemp" := "ContadorSimi"; END_IF;
   #_w12 := #_w9 AND NOT "BloqueoSimilares4" AND ("Var".VectorPrincipalJ1["IntentoCompletoJ1", 1] <> "Var".CodigoOJ1[1]);
   IF #_w12 AND ("Var".VectorPrincipalJ1["IntentoCompletoJ1", 1] = "Var".CodigoSimilaresJ1[0]) THEN
       "BloqueoSimilares1" := TRUE;
   END_IF;
   #_w13 := #_w12 AND ("Var".VectorPrincipalJ1["IntentoCompletoJ1", 1] <> "Var".CodigoSimilaresJ1[0]);
   IF #_w13 AND ("Var".VectorPrincipalJ1["IntentoCompletoJ1", 1] = "Var".CodigoSimilaresJ1[2]) THEN
       "BloqueoSimilares2" := TRUE;
   END_IF;
   IF #_w13 AND ("Var".VectorPrincipalJ1["IntentoCompletoJ1", 1] <> "Var".CodigoSimilaresJ1[2]) AND ("Var".VectorPrincipalJ1["IntentoCompletoJ1", 1] = "Var".CodigoSimilaresJ1[3]) THEN
       "BloqueoSimilares3" := TRUE;
   END_IF;
   #_w14 := #_w9 AND "BloqueoSimilares1";
   IF #_w14 THEN "Var".CodigoSimilaresJ1[0] := 8; END_IF;
   "ContadorSimilares".CTU(CU := #_w14, R := "ReiniciarChecarSimi", PV := 3, CV => "ContadorSimi");
   IF #_w14 THEN
       "ContadorSimiTemp" := "ContadorSimi";
       "BloqueoSimilares1" := FALSE;
   END_IF;
   #_w15 := #_w9 AND "BloqueoSimilares2";
   IF #_w15 THEN "Var".CodigoSimilaresJ1[2] := 8; END_IF;
   "ContadorSimilares".CTU(CU := #_w15, R := "ReiniciarChecarSimi", PV := 3, CV => "ContadorSimi");
   IF #_w15 THEN
       "ContadorSimiTemp" := "ContadorSimi";
       "BloqueoSimilares2" := FALSE;
   END_IF;
   #_w16 := #_w9 AND "BloqueoSimilares3";
   IF #_w16 THEN "Var".CodigoSimilaresJ1[3] := 8; END_IF;
   "ContadorSimilares".CTU(CU := #_w16, R := "ReiniciarChecarSimi", PV := 3, CV => "ContadorSimi");
   IF #_w16 THEN
       "ContadorSimiTemp" := "ContadorSimi";
       "BloqueoSimilares3" := FALSE;
   END_IF;
   #_w17 := "Panel1AmarilloJ1" AND "Bounce3" AND "Panel1AmarilloJ1" AND "Intento1J1" AND ("Var".VectorPrincipalJ1["IntentoCompletoJ1", 2] = 0);
   IF #_w17 THEN
       "Var".VectorPrincipalJ1["IntentoCompletoJ1", 2] := 7;
       "Intento2J1" := TRUE;
   END_IF;
   #_w18 := #_w17 AND ("Var".VectorPrincipalJ1["IntentoCompletoJ1", 2] = "Var".CodigoOJ1[2]);
   "ContadorCorrectas".CTU(CU := #_w18, R := "ReiniciarChecarCorr", PV := 3, CV => "ContadorCorr");
   IF #_w18 THEN
       "ContadorCorrTemp" := "ContadorCorr";
       "Var".CodigoSimilaresJ1[2] := 8;
       "BloqueoSimilares4" := TRUE;
   END_IF;
   #_w19 := #_w18 AND ("Var".CodigoSimilaresJ1[2] = 8);
   "ContadorSimilares".CTD(CD := #_w19, LD := "ReiniciarChecarSimi", PV := 3, CV => "ContadorSimi");
   IF #_w19 THEN "ContadorSimiTemp" := "ContadorSimi"; END_IF;
   #_w20 := #_w17 AND NOT "BloqueoSimilares4" AND ("Var".VectorPrincipalJ1["IntentoCompletoJ1", 2] <> "Var".CodigoOJ1[2]);
   IF #_w20 AND ("Var".VectorPrincipalJ1["IntentoCompletoJ1", 2] = "Var".CodigoSimilaresJ1[0]) THEN
       "BloqueoSimilares1" := TRUE;
   END_IF;
   #_w21 := #_w20 AND ("Var".VectorPrincipalJ1["IntentoCompletoJ1", 2] <> "Var".CodigoSimilaresJ1[0]);
   IF #_w21 AND ("Var".VectorPrincipalJ1["IntentoCompletoJ1", 2] = "Var".CodigoSimilaresJ1[1]) THEN
       "BloqueoSimilares2" := TRUE;
   END_IF;
   IF #_w21 AND ("Var".VectorPrincipalJ1["IntentoCompletoJ1", 2] <> "Var".CodigoSimilaresJ1[1]) AND ("Var".VectorPrincipalJ1["IntentoCompletoJ1", 2] = "Var".CodigoSimilaresJ1[3]) THEN
       "BloqueoSimilares3" := TRUE;
   END_IF;
   #_w22 := #_w17 AND "BloqueoSimilares1";
   IF #_w22 THEN "Var".CodigoSimilaresJ1[0] := 8; END_IF;
   "ContadorSimilares".CTU(CU := #_w22, R := "ReiniciarChecarSimi", PV := 3, CV => "ContadorSimi");
   IF #_w22 THEN
       "ContadorSimiTemp" := "ContadorSimi";
       "BloqueoSimilares1" := FALSE;
   END_IF;
   #_w23 := #_w17 AND "BloqueoSimilares2";
   IF #_w23 THEN "Var".CodigoSimilaresJ1[1] := 8; END_IF;
   "ContadorSimilares".CTU(CU := #_w23, R := "ReiniciarChecarSimi", PV := 3, CV => "ContadorSimi");
   IF #_w23 THEN
       "ContadorSimiTemp" := "ContadorSimi";
       "BloqueoSimilares2" := FALSE;
   END_IF;
   #_w24 := #_w17 AND "BloqueoSimilares3";
   IF #_w24 THEN "Var".CodigoSimilaresJ1[3] := 8; END_IF;
   "ContadorSimilares".CTU(CU := #_w24, R := "ReiniciarChecarSimi", PV := 3, CV => "ContadorSimi");
   IF #_w24 THEN
       "ContadorSimiTemp" := "ContadorSimi";
       "BloqueoSimilares3" := FALSE;
   END_IF;
   #_w25 := "Panel1AmarilloJ1" AND "Bounce4" AND "Panel1AmarilloJ1" AND "Intento2J1" AND ("Var".VectorPrincipalJ1["IntentoCompletoJ1", 3] = 0);
   IF #_w25 THEN
       "Var".VectorPrincipalJ1["IntentoCompletoJ1", 3] := 7;
       "Intento3J1" := TRUE;
   END_IF;
   #_w26 := #_w25 AND ("Var".VectorPrincipalJ1["IntentoCompletoJ1", 3] = "Var".CodigoOJ1[3]);
   "ContadorCorrectas".CTU(CU := #_w26, R := "ReiniciarChecarCorr", PV := 3, CV => "ContadorCorr");
   IF #_w26 THEN
       "ContadorCorrTemp" := "ContadorCorr";
       "Var".CodigoSimilaresJ1[3] := 8;
       "BloqueoSimilares4" := TRUE;
   END_IF;
   #_w27 := #_w26 AND ("Var".CodigoSimilaresJ1[3] = 8);
   "ContadorSimilares".CTD(CD := #_w27, LD := "ReiniciarChecarSimi", PV := 3, CV => "ContadorSimi");
   IF #_w27 THEN "ContadorSimiTemp" := "ContadorSimi"; END_IF;
   #_w28 := #_w25 AND NOT "BloqueoSimilares4" AND ("Var".VectorPrincipalJ1["IntentoCompletoJ1", 3] <> "Var".CodigoOJ1[3]);
   IF #_w28 AND ("Var".VectorPrincipalJ1["IntentoCompletoJ1", 3] = "Var".CodigoSimilaresJ1[0]) THEN
       "BloqueoSimilares1" := TRUE;
   END_IF;
   #_w29 := #_w28 AND ("Var".VectorPrincipalJ1["IntentoCompletoJ1", 3] <> "Var".CodigoSimilaresJ1[0]);
   IF #_w29 AND ("Var".VectorPrincipalJ1["IntentoCompletoJ1", 3] = "Var".CodigoSimilaresJ1[1]) THEN
       "BloqueoSimilares2" := TRUE;
   END_IF;
   IF #_w29 AND ("Var".VectorPrincipalJ1["IntentoCompletoJ1", 3] <> "Var".CodigoSimilaresJ1[1]) AND ("Var".VectorPrincipalJ1["IntentoCompletoJ1", 3] = "Var".CodigoSimilaresJ1[2]) THEN
       "BloqueoSimilares3" := TRUE;
   END_IF;
   #_w30 := #_w25 AND "BloqueoSimilares1";
   IF #_w30 THEN "Var".CodigoSimilaresJ1[0] := 8; END_IF;
   "ContadorSimilares".CTU(CU := #_w30, R := "ReiniciarChecarSimi", PV := 3, CV => "ContadorSimi");
   IF #_w30 THEN
       "ContadorSimiTemp" := "ContadorSimi";
       "BloqueoSimilares1" := FALSE;
   END_IF;
   #_w31 := #_w25 AND "BloqueoSimilares2";
   IF #_w31 THEN "Var".CodigoSimilaresJ1[1] := 8; END_IF;
   "ContadorSimilares".CTU(CU := #_w31, R := "ReiniciarChecarSimi", PV := 3, CV => "ContadorSimi");
   IF #_w31 THEN
       "ContadorSimiTemp" := "ContadorSimi";
       "BloqueoSimilares2" := FALSE;
   END_IF;
   #_w32 := #_w25 AND "BloqueoSimilares3";
   IF #_w32 THEN "Var".CodigoSimilaresJ1[2] := 8; END_IF;
   "ContadorSimilares".CTU(CU := #_w32, R := "ReiniciarChecarSimi", PV := 3, CV => "ContadorSimi");
   IF #_w32 THEN
       "ContadorSimiTemp" := "ContadorSimi";
       "BloqueoSimilares3" := FALSE;
   END_IF;
END_REGION

REGION Network 13: Comprobar Intentos
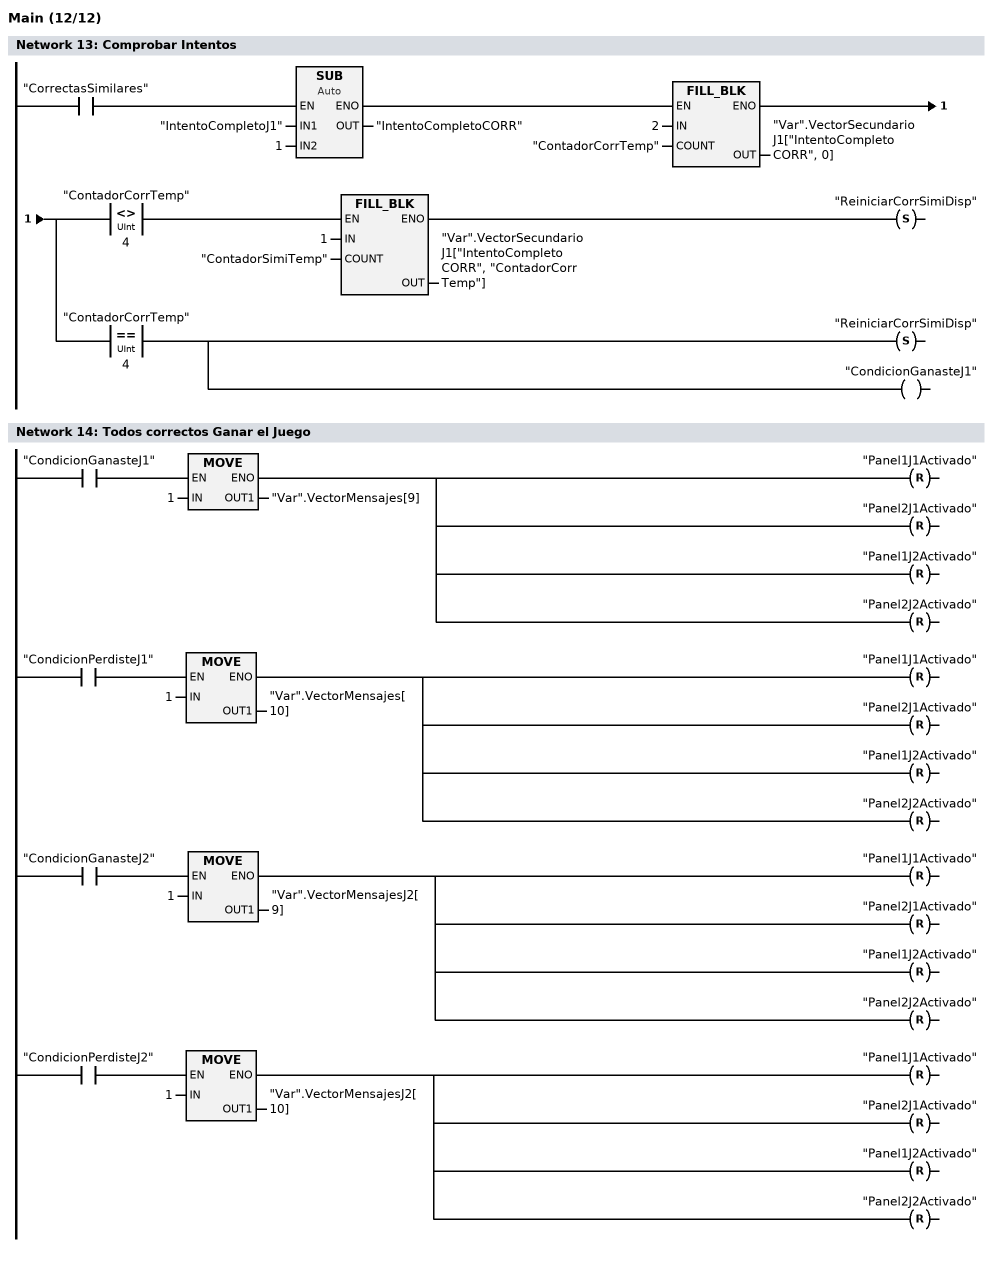
   RUNG wire#powerrail
      Contact( "CorrectasSimilares" )
      Sub(in1 := "IntentoCompletoJ1", in2 := 1, out => "IntentoCompletoCORR")
      FillBlockI(in := 2, count := "ContadorCorrTemp", out => "Var".VectorSecundarioJ1["IntentoCompletoCORR", 0])
      wire#w1
      { S7_Templates := "SrcType := UInt" } NE_Contact(in1 := "ContadorCorrTemp", in2 := 4)
      FillBlockI(in := 1, count := "ContadorSimiTemp", out => "Var".VectorSecundarioJ1["IntentoCompletoCORR", "ContadorCorrTemp"])
      S_Coil( "ReiniciarCorrSimiDisp" )
   END_RUNG
   RUNG wire#w1
      { S7_Templates := "SrcType := UInt" } EQ_Contact(in1 := "ContadorCorrTemp", in2 := 4)
      wire#w2
      S_Coil( "ReiniciarCorrSimiDisp" )
   END_RUNG
   RUNG wire#w2
      Coil( "CondicionGanasteJ1" )
   END_RUNG
   // the same network as SCL:
   IF "CorrectasSimilares" THEN "IntentoCompletoCORR" := "IntentoCompletoJ1" - 1; END_IF;
   #_w1 := "CorrectasSimilares";
   IF #_w1 THEN
       FILL_BLK(IN := 2, COUNT := "ContadorCorrTemp", OUT => "Var".VectorSecundarioJ1["IntentoCompletoCORR", 0]);
   END_IF;
   #_w2 := #_w1 AND ("ContadorCorrTemp" <> 4);
   IF #_w2 THEN
       FILL_BLK(IN := 1,
                COUNT := "ContadorSimiTemp",
                OUT => "Var".VectorSecundarioJ1["IntentoCompletoCORR", "ContadorCorrTemp"]);
       "ReiniciarCorrSimiDisp" := TRUE;
   END_IF;
   #_w3 := #_w1 AND ("ContadorCorrTemp" = 4);
   IF #_w3 THEN "ReiniciarCorrSimiDisp" := TRUE; END_IF;
   "CondicionGanasteJ1" := #_w3;
END_REGION

REGION Network 14: Todos correctos Ganar el Juego
   RUNG wire#powerrail
      Contact( "CondicionGanasteJ1" )
      Move(in := 1, out1 => "Var".VectorMensajes[9])
      wire#w1
      R_Coil( "Panel1J1Activado" )
   END_RUNG
   RUNG wire#w1
      R_Coil( "Panel2J1Activado" )
   END_RUNG
   RUNG wire#w1
      R_Coil( "Panel1J2Activado" )
   END_RUNG
   RUNG wire#w1
      R_Coil( "Panel2J2Activado" )
   END_RUNG
   RUNG wire#powerrail
      Contact( "CondicionPerdisteJ1" )
      Move(in := 1, out1 => "Var".VectorMensajes[10])
      wire#w2
      R_Coil( "Panel1J1Activado" )
   END_RUNG
   RUNG wire#w2
      R_Coil( "Panel2J1Activado" )
   END_RUNG
   RUNG wire#w2
      R_Coil( "Panel1J2Activado" )
   END_RUNG
   RUNG wire#w2
      R_Coil( "Panel2J2Activado" )
   END_RUNG
   RUNG wire#powerrail
      Contact( "CondicionGanasteJ2" )
      Move(in := 1, out1 => "Var".VectorMensajesJ2[9])
      wire#w3
      R_Coil( "Panel1J1Activado" )
   END_RUNG
   RUNG wire#w3
      R_Coil( "Panel2J1Activado" )
   END_RUNG
   RUNG wire#w3
      R_Coil( "Panel1J2Activado" )
   END_RUNG
   RUNG wire#w3
      R_Coil( "Panel2J2Activado" )
   END_RUNG
   RUNG wire#powerrail
      Contact( "CondicionPerdisteJ2" )
      Move(in := 1, out1 => "Var".VectorMensajesJ2[10])
      wire#w4
      R_Coil( "Panel1J1Activado" )
   END_RUNG
   RUNG wire#w4
      R_Coil( "Panel2J1Activado" )
   END_RUNG
   RUNG wire#w4
      R_Coil( "Panel1J2Activado" )
   END_RUNG
   RUNG wire#w4
      R_Coil( "Panel2J2Activado" )
   END_RUNG
   // the same network as SCL:
   IF "CondicionGanasteJ1" THEN
       "Var".VectorMensajes[9] := 1;
       "Panel1J1Activado" := FALSE;
       "Panel2J1Activado" := FALSE;
       "Panel1J2Activado" := FALSE;
       "Panel2J2Activado" := FALSE;
   END_IF;
   IF "CondicionPerdisteJ1" THEN
       "Var".VectorMensajes[10] := 1;
       "Panel1J1Activado" := FALSE;
       "Panel2J1Activado" := FALSE;
       "Panel1J2Activado" := FALSE;
       "Panel2J2Activado" := FALSE;
   END_IF;
   IF "CondicionGanasteJ2" THEN
       "Var".VectorMensajesJ2[9] := 1;
       "Panel1J1Activado" := FALSE;
       "Panel2J1Activado" := FALSE;
       "Panel1J2Activado" := FALSE;
       "Panel2J2Activado" := FALSE;
   END_IF;
   IF "CondicionPerdisteJ2" THEN
       "Var".VectorMensajesJ2[10] := 1;
       "Panel1J1Activado" := FALSE;
       "Panel2J1Activado" := FALSE;
       "Panel1J2Activado" := FALSE;
       "Panel2J2Activado" := FALSE;
   END_IF;
END_REGION
END_ORGANIZATION_BLOCK

(* ===== HMI "HMI_RT_1" =====
system functions are stored by id; their names below are inferred from use
connection "HMI_Connection_1": ETHERNET, S7_1500_OMS

HMI tags "Default tag table"
   "Tag_ScreenNumber" : UInt, internal
   "ReiniciarJuego" : Bool = PLC ReiniciarJuego AT %M6.0, 1 s
   "Panel2CafeJ1" : Bool = PLC Panel2CafeJ1 AT %M10.4, 1 s
   "Panel2RosaJ1" : Bool = PLC Panel2RosaJ1 AT %M10.5, 1 s
   "Panel2MoradoJ1" : Bool = PLC Panel2MoradoJ1 AT %M10.6, 1 s
   "Panel2RojoJ1" : Bool = PLC Panel2RojoJ1 AT %M10.7, 1 s
   "Panel2AzulJ1" : Bool = PLC Panel2AzulJ1 AT %M11.0, 1 s
   "Panel2VerdeJ1" : Bool = PLC Panel2VerdeJ1 AT %M11.1, 1 s
   "Panel2AmarilloJ1" : Bool = PLC Panel2AmarilloJ1 AT %M11.2, 1 s
   "Panel1CafeJ1" : Bool = PLC Panel1CafeJ1 AT %M9.5, 1 s
   "Panel1RosaJ1" : Bool = PLC Panel1RosaJ1 AT %M9.6, 1 s
   "Panel1MoradoJ1" : Bool = PLC Panel1MoradoJ1 AT %M9.7, 1 s
   "Panel1RojoJ1" : Bool = PLC Panel1RojoJ1 AT %M10.0, 1 s
   "Panel1AzulJ1" : Bool = PLC Panel1AzulJ1 AT %M10.1, 1 s
   "Panel1VerdeJ1" : Bool = PLC Panel1VerdeJ1 AT %M10.2, 1 s
   "Panel1AmarilloJ1" : Bool = PLC Panel1AmarilloJ1 AT %M10.3, 1 s
   "Panel1J1Activado" : Bool = PLC Panel1J1Activado AT %M13.1, 1 s
   "Panel2J1Activado" : Bool = PLC Panel2J1Activado AT %M13.2, 1 s
   "Var_VectorMensajes{0}" : Int = PLC "Var".VectorMensajes[0], 1 s
   "Var_VectorMensajes{1}" : Int = PLC "Var".VectorMensajes[1], 1 s
   "Var_VectorMensajes{2}" : Int = PLC "Var".VectorMensajes[2], 1 s
   "Var_VectorMensajes{3}" : Int = PLC "Var".VectorMensajes[3], 1 s
   "Var_VectorMensajes{4}" : Int = PLC "Var".VectorMensajes[4], 1 s
   "Var_VectorMensajes{5}" : Int = PLC "Var".VectorMensajes[5], 1 s
   "Var_VectorMensajes{6}" : Int = PLC "Var".VectorMensajes[6], 1 s
   "Var_VectorMensajes{7}" : Int = PLC "Var".VectorMensajes[7], 1 s
   "Var_VectorMensajes{8}" : Int = PLC "Var".VectorMensajes[8], 1 s
   "Var_VectorMensajes{9}" : Int = PLC "Var".VectorMensajes[9], 1 s
   "Var_VectorMensajes{10}" : Int = PLC "Var".VectorMensajes[10], 1 s
   "Var_CodigoOJ1{0}" : Int = PLC "Var".CodigoOJ1[0], 1 s
   "Var_CodigoOJ1{1}" : Int = PLC "Var".CodigoOJ1[1], 1 s
   "Var_CodigoOJ1{2}" : Int = PLC "Var".CodigoOJ1[2], 1 s
   "Var_CodigoOJ1{3}" : Int = PLC "Var".CodigoOJ1[3], 1 s
   "Var_CodigoSJ1{0}" : Int = PLC "Var".CodigoSJ1[0], 1 s
   "Var_CodigoSJ1{1}" : Int = PLC "Var".CodigoSJ1[1], 1 s
   "Var_CodigoSJ1{2}" : Int = PLC "Var".CodigoSJ1[2], 1 s
   "Var_CodigoSJ1{3}" : Int = PLC "Var".CodigoSJ1[3], 1 s
   "Var_VectorPrincipalJ1{0,0}" : Int = PLC "Var".VectorPrincipalJ1[0,0], 1 s
   "Var_VectorPrincipalJ1{0,1}" : Int = PLC "Var".VectorPrincipalJ1[0,1], 1 s
   "Var_VectorPrincipalJ1{0,2}" : Int = PLC "Var".VectorPrincipalJ1[0,2], 1 s
   "Var_VectorPrincipalJ1{0,3}" : Int = PLC "Var".VectorPrincipalJ1[0,3], 1 s
   "Var_VectorPrincipalJ1{1,0}" : Int = PLC "Var".VectorPrincipalJ1[1,0], 1 s
   "Var_VectorPrincipalJ1{1,1}" : Int = PLC "Var".VectorPrincipalJ1[1,1], 1 s
   "Var_VectorPrincipalJ1{1,2}" : Int = PLC "Var".VectorPrincipalJ1[1,2], 1 s
   "Var_VectorPrincipalJ1{1,3}" : Int = PLC "Var".VectorPrincipalJ1[1,3], 1 s
   "Var_VectorPrincipalJ1{2,0}" : Int = PLC "Var".VectorPrincipalJ1[2,0], 1 s
   "Var_VectorPrincipalJ1{2,1}" : Int = PLC "Var".VectorPrincipalJ1[2,1], 1 s
   "Var_VectorPrincipalJ1{2,2}" : Int = PLC "Var".VectorPrincipalJ1[2,2], 1 s
   "Var_VectorPrincipalJ1{2,3}" : Int = PLC "Var".VectorPrincipalJ1[2,3], 1 s
   "Var_VectorPrincipalJ1{3,0}" : Int = PLC "Var".VectorPrincipalJ1[3,0], 1 s
   "Var_VectorPrincipalJ1{3,1}" : Int = PLC "Var".VectorPrincipalJ1[3,1], 1 s
   "Var_VectorPrincipalJ1{3,2}" : Int = PLC "Var".VectorPrincipalJ1[3,2], 1 s
   "Var_VectorPrincipalJ1{3,3}" : Int = PLC "Var".VectorPrincipalJ1[3,3], 1 s
   "Var_VectorPrincipalJ1{4,0}" : Int = PLC "Var".VectorPrincipalJ1[4,0], 1 s
   "Var_VectorPrincipalJ1{4,1}" : Int = PLC "Var".VectorPrincipalJ1[4,1], 1 s
   "Var_VectorPrincipalJ1{4,2}" : Int = PLC "Var".VectorPrincipalJ1[4,2], 1 s
   "Var_VectorPrincipalJ1{4,3}" : Int = PLC "Var".VectorPrincipalJ1[4,3], 1 s
   "Var_VectorPrincipalJ1{5,0}" : Int = PLC "Var".VectorPrincipalJ1[5,0], 1 s
   "Var_VectorPrincipalJ1{5,1}" : Int = PLC "Var".VectorPrincipalJ1[5,1], 1 s
   "Var_VectorPrincipalJ1{5,2}" : Int = PLC "Var".VectorPrincipalJ1[5,2], 1 s
   "Var_VectorPrincipalJ1{5,3}" : Int = PLC "Var".VectorPrincipalJ1[5,3], 1 s
   "Var_VectorPrincipalJ1{6,0}" : Int = PLC "Var".VectorPrincipalJ1[6,0], 1 s
   "Var_VectorPrincipalJ1{6,1}" : Int = PLC "Var".VectorPrincipalJ1[6,1], 1 s
   "Var_VectorPrincipalJ1{6,2}" : Int = PLC "Var".VectorPrincipalJ1[6,2], 1 s
   "Var_VectorPrincipalJ1{6,3}" : Int = PLC "Var".VectorPrincipalJ1[6,3], 1 s
   "Var_VectorPrincipalJ1{7,0}" : Int = PLC "Var".VectorPrincipalJ1[7,0], 1 s
   "Var_VectorPrincipalJ1{7,1}" : Int = PLC "Var".VectorPrincipalJ1[7,1], 1 s
   "Var_VectorPrincipalJ1{7,2}" : Int = PLC "Var".VectorPrincipalJ1[7,2], 1 s
   "Var_VectorPrincipalJ1{7,3}" : Int = PLC "Var".VectorPrincipalJ1[7,3], 1 s
   "Var_VectorSecundarioJ1{0,0}" : Int = PLC "Var".VectorSecundarioJ1[0,0], 1 s
   "Var_VectorSecundarioJ1{0,1}" : Int = PLC "Var".VectorSecundarioJ1[0,1], 1 s
   "Var_VectorSecundarioJ1{0,2}" : Int = PLC "Var".VectorSecundarioJ1[0,2], 1 s
   "Var_VectorSecundarioJ1{0,3}" : Int = PLC "Var".VectorSecundarioJ1[0,3], 1 s
   "Var_VectorSecundarioJ1{1,0}" : Int = PLC "Var".VectorSecundarioJ1[1,0], 1 s
   "Var_VectorSecundarioJ1{1,1}" : Int = PLC "Var".VectorSecundarioJ1[1,1], 1 s
   "Var_VectorSecundarioJ1{1,2}" : Int = PLC "Var".VectorSecundarioJ1[1,2], 1 s
   "Var_VectorSecundarioJ1{1,3}" : Int = PLC "Var".VectorSecundarioJ1[1,3], 1 s
   "Var_VectorSecundarioJ1{2,0}" : Int = PLC "Var".VectorSecundarioJ1[2,0], 1 s
   "Var_VectorSecundarioJ1{2,1}" : Int = PLC "Var".VectorSecundarioJ1[2,1], 1 s
   "Var_VectorSecundarioJ1{2,2}" : Int = PLC "Var".VectorSecundarioJ1[2,2], 1 s
   "Var_VectorSecundarioJ1{2,3}" : Int = PLC "Var".VectorSecundarioJ1[2,3], 1 s
   "Var_VectorSecundarioJ1{3,0}" : Int = PLC "Var".VectorSecundarioJ1[3,0], 1 s
   "Var_VectorSecundarioJ1{3,1}" : Int = PLC "Var".VectorSecundarioJ1[3,1], 1 s
   "Var_VectorSecundarioJ1{3,2}" : Int = PLC "Var".VectorSecundarioJ1[3,2], 1 s
   "Var_VectorSecundarioJ1{3,3}" : Int = PLC "Var".VectorSecundarioJ1[3,3], 1 s
   "Var_VectorSecundarioJ1{4,0}" : Int = PLC "Var".VectorSecundarioJ1[4,0], 1 s
   "Var_VectorSecundarioJ1{4,1}" : Int = PLC "Var".VectorSecundarioJ1[4,1], 1 s
   "Var_VectorSecundarioJ1{4,2}" : Int = PLC "Var".VectorSecundarioJ1[4,2], 1 s
   "Var_VectorSecundarioJ1{4,3}" : Int = PLC "Var".VectorSecundarioJ1[4,3], 1 s
   "Var_VectorSecundarioJ1{5,0}" : Int = PLC "Var".VectorSecundarioJ1[5,0], 1 s
   "Var_VectorSecundarioJ1{5,1}" : Int = PLC "Var".VectorSecundarioJ1[5,1], 1 s
   "Var_VectorSecundarioJ1{5,2}" : Int = PLC "Var".VectorSecundarioJ1[5,2], 1 s
   "Var_VectorSecundarioJ1{5,3}" : Int = PLC "Var".VectorSecundarioJ1[5,3], 1 s
   "Var_VectorSecundarioJ1{6,0}" : Int = PLC "Var".VectorSecundarioJ1[6,0], 1 s
   "Var_VectorSecundarioJ1{6,1}" : Int = PLC "Var".VectorSecundarioJ1[6,1], 1 s
   "Var_VectorSecundarioJ1{6,2}" : Int = PLC "Var".VectorSecundarioJ1[6,2], 1 s
   "Var_VectorSecundarioJ1{6,3}" : Int = PLC "Var".VectorSecundarioJ1[6,3], 1 s
   "Var_VectorSecundarioJ1{7,0}" : Int = PLC "Var".VectorSecundarioJ1[7,0], 1 s
   "Var_VectorSecundarioJ1{7,1}" : Int = PLC "Var".VectorSecundarioJ1[7,1], 1 s
   "Var_VectorSecundarioJ1{7,2}" : Int = PLC "Var".VectorSecundarioJ1[7,2], 1 s
   "Var_VectorSecundarioJ1{7,3}" : Int = PLC "Var".VectorSecundarioJ1[7,3], 1 s
   "Bounce1" : Bool = PLC Bounce1 AT %M13.6, 1 s
   "Bounce5" : Bool = PLC Bounce5 AT %M14.1, 1 s
   "ReiniciarCorrSimiDisp" : Bool = PLC ReiniciarCorrSimiDisp AT %M34.0, 1 s

screen "Root screen" 800x442, template "Template_1"
   on GenerateScreen: SetTag("Tag_ScreenNumber", 1)
   Button "Button_3" at 67,293 size 28x26; TextOff 'Text'
      on Press: SetBit("Panel1CafeJ1")
      on Release: SetBit("Bounce5"); ResetBit("Panel1CafeJ1")
      Appearance <- "Panel1J1Activado"
   Button "Button_4" at 99,293 size 27x26; TextOff 'Text'
      on Press: SetBit("Panel1RosaJ1")
      on Release: SetBit("Bounce5"); ResetBit("Panel1RosaJ1")
      Appearance <- "Panel1J1Activado"
   Button "Button_5" at 131,293 size 27x24; TextOff 'Text'
      on Press: SetBit("Panel1MoradoJ1")
      on Release: SetBit("Bounce5"); ResetBit("Panel1MoradoJ1")
      Appearance <- "Panel1J1Activado"
   Button "Button_6" at 165,293 size 25x25; TextOff 'Text'
      on Press: SetBit("Panel1RojoJ1")
      on Release: SetBit("Bounce5"); ResetBit("Panel1RojoJ1")
      Appearance <- "Panel1J1Activado"
   Button "Button_7" at 196,293 size 25x24; TextOff 'Text'
      on Press: SetBit("Panel1AzulJ1")
      on Release: SetBit("Bounce5"); ResetBit("Panel1AzulJ1")
      Appearance <- "Panel1J1Activado"
   Button "Button_8" at 227,293 size 25x25; TextOff 'Text'
      on Press: SetBit("Panel1VerdeJ1")
      on Release: SetBit("Bounce5"); ResetBit("Panel1VerdeJ1")
      Appearance <- "Panel1J1Activado"
   Button "Button_9" at 256,294 size 25x23; TextOff 'Text'
      on Press: SetBit("Panel1AmarilloJ1")
      on Release: SetBit("Bounce5"); ResetBit("Panel1AmarilloJ1")
      Appearance <- "Panel1J1Activado"
   TextField "Text field_1" at 37,250 size 16x23; Text '1'
   TextField "Text field_2" at 37,221 size 16x23; Text '2'
   TextField "Text field_3" at 37,194 size 16x23; Text '3'
   TextField "Text field_4" at 37,163 size 16x23; Text '4'
   TextField "Text field_5" at 37,134 size 16x23; Text '5'
   TextField "Text field_6" at 37,103 size 16x23; Text '6'
   TextField "Text field_7" at 37,74 size 16x23; Text '7'
   TextField "Text field_8" at 37,43 size 16x23; Text '8'
   Circle "Circle_1" at 92,254 size 23x23
      Appearance <- "Var_VectorPrincipalJ1{0,0}"
   Circle "Circle_2" at 128,254 size 23x23
      Appearance <- "Var_VectorPrincipalJ1{0,1}"
   Circle "Circle_3" at 164,254 size 23x23
      Appearance <- "Var_VectorPrincipalJ1{0,2}"
   Circle "Circle_4" at 201,254 size 23x23
      Appearance <- "Var_VectorPrincipalJ1{0,3}"
   Circle "Circle_5" at 92,224 size 23x23
      Appearance <- "Var_VectorPrincipalJ1{1,0}"
   Circle "Circle_6" at 128,224 size 23x23
      Appearance <- "Var_VectorPrincipalJ1{1,1}"
   Circle "Circle_7" at 164,224 size 23x23
      Appearance <- "Var_VectorPrincipalJ1{1,2}"
   Circle "Circle_8" at 201,224 size 23x23
      Appearance <- "Var_VectorPrincipalJ1{1,3}"
   Circle "Circle_9" at 92,194 size 23x23
      Appearance <- "Var_VectorPrincipalJ1{2,0}"
   Circle "Circle_10" at 128,194 size 23x23
      Appearance <- "Var_VectorPrincipalJ1{2,1}"
   Circle "Circle_11" at 164,194 size 23x23
      Appearance <- "Var_VectorPrincipalJ1{2,2}"
   Circle "Circle_12" at 201,194 size 23x23
      Appearance <- "Var_VectorPrincipalJ1{2,3}"
   Circle "Circle_13" at 92,164 size 23x23
      Appearance <- "Var_VectorPrincipalJ1{3,0}"
   Circle "Circle_14" at 128,164 size 23x23
      Appearance <- "Var_VectorPrincipalJ1{3,1}"
   Circle "Circle_15" at 164,164 size 23x23
      Appearance <- "Var_VectorPrincipalJ1{3,2}"
   Circle "Circle_16" at 201,164 size 23x23
      Appearance <- "Var_VectorPrincipalJ1{3,3}"
   Circle "Circle_17" at 92,134 size 23x23
      Appearance <- "Var_VectorPrincipalJ1{4,0}"
   Circle "Circle_18" at 128,134 size 23x23
      Appearance <- "Var_VectorPrincipalJ1{4,1}"
   Circle "Circle_19" at 164,134 size 23x23
      Appearance <- "Var_VectorPrincipalJ1{4,2}"
   Circle "Circle_20" at 201,134 size 23x23
      Appearance <- "Var_VectorPrincipalJ1{4,3}"
   Circle "Circle_21" at 92,104 size 23x23
      Appearance <- "Var_VectorPrincipalJ1{5,0}"
   Circle "Circle_22" at 128,104 size 23x23
      Appearance <- "Var_VectorPrincipalJ1{5,1}"
   Circle "Circle_23" at 164,104 size 23x23
      Appearance <- "Var_VectorPrincipalJ1{5,2}"
   Circle "Circle_24" at 201,104 size 23x23
      Appearance <- "Var_VectorPrincipalJ1{5,3}"
   Circle "Circle_25" at 92,74 size 23x23
      Appearance <- "Var_VectorPrincipalJ1{6,0}"
   Circle "Circle_26" at 128,74 size 23x23
      Appearance <- "Var_VectorPrincipalJ1{6,1}"
   Circle "Circle_27" at 164,74 size 23x23
      Appearance <- "Var_VectorPrincipalJ1{6,2}"
   Circle "Circle_28" at 201,74 size 23x23
      Appearance <- "Var_VectorPrincipalJ1{6,3}"
   Circle "Circle_29" at 92,44 size 23x23
      Appearance <- "Var_VectorPrincipalJ1{7,0}"
   Circle "Circle_30" at 128,44 size 23x23
      Appearance <- "Var_VectorPrincipalJ1{7,1}"
   Circle "Circle_31" at 164,44 size 23x23
      Appearance <- "Var_VectorPrincipalJ1{7,2}"
   Circle "Circle_32" at 201,44 size 23x23
      Appearance <- "Var_VectorPrincipalJ1{7,3}"
   Circle "Circle_33" at 255,253 size 14x14
      Appearance <- "Var_VectorSecundarioJ1{0,0}"
   Circle "Circle_34" at 270,253 size 14x14
      Appearance <- "Var_VectorSecundarioJ1{0,1}"
   Circle "Circle_35" at 255,267 size 14x14
      Appearance <- "Var_VectorSecundarioJ1{0,2}"
   Circle "Circle_36" at 270,267 size 14x14
      Appearance <- "Var_VectorSecundarioJ1{0,3}"
   Circle "Circle_37" at 255,223 size 14x14
      Appearance <- "Var_VectorSecundarioJ1{1,0}"
   Circle "Circle_38" at 270,223 size 14x14
      Appearance <- "Var_VectorSecundarioJ1{1,1}"
   Circle "Circle_39" at 255,237 size 14x14
      Appearance <- "Var_VectorSecundarioJ1{1,2}"
   Circle "Circle_40" at 270,237 size 14x14
      Appearance <- "Var_VectorSecundarioJ1{1,3}"
   Circle "Circle_41" at 255,193 size 14x14
      Appearance <- "Var_VectorSecundarioJ1{2,0}"
   Circle "Circle_42" at 270,193 size 14x14
      Appearance <- "Var_VectorSecundarioJ1{2,1}"
   Circle "Circle_43" at 255,207 size 14x14
      Appearance <- "Var_VectorSecundarioJ1{2,2}"
   Circle "Circle_44" at 270,207 size 14x14
      Appearance <- "Var_VectorSecundarioJ1{2,3}"
   Circle "Circle_45" at 255,163 size 14x14
      Appearance <- "Var_VectorSecundarioJ1{3,0}"
   Circle "Circle_46" at 270,163 size 14x14
      Appearance <- "Var_VectorSecundarioJ1{3,1}"
   Circle "Circle_47" at 255,177 size 14x14
      Appearance <- "Var_VectorSecundarioJ1{3,2}"
   Circle "Circle_48" at 270,177 size 14x14
      Appearance <- "Var_VectorSecundarioJ1{3,3}"
   Circle "Circle_49" at 255,133 size 14x14
      Appearance <- "Var_VectorSecundarioJ1{4,0}"
   Circle "Circle_50" at 270,133 size 14x14
      Appearance <- "Var_VectorSecundarioJ1{4,1}"
   Circle "Circle_51" at 255,147 size 14x14
      Appearance <- "Var_VectorSecundarioJ1{4,2}"
   Circle "Circle_52" at 270,147 size 14x14
      Appearance <- "Var_VectorSecundarioJ1{4,3}"
   Circle "Circle_53" at 255,103 size 14x14
      Appearance <- "Var_VectorSecundarioJ1{5,0}"
   Circle "Circle_54" at 270,103 size 14x14
      Appearance <- "Var_VectorSecundarioJ1{5,1}"
   Circle "Circle_55" at 255,117 size 14x14
      Appearance <- "Var_VectorSecundarioJ1{5,2}"
   Circle "Circle_56" at 270,117 size 14x14
      Appearance <- "Var_VectorSecundarioJ1{5,3}"
   Circle "Circle_57" at 255,73 size 14x14
      Appearance <- "Var_VectorSecundarioJ1{6,0}"
   Circle "Circle_58" at 270,73 size 14x14
      Appearance <- "Var_VectorSecundarioJ1{6,1}"
   Circle "Circle_59" at 255,87 size 14x14
      Appearance <- "Var_VectorSecundarioJ1{6,2}"
   Circle "Circle_60" at 270,87 size 14x14
      Appearance <- "Var_VectorSecundarioJ1{6,3}"
   Circle "Circle_61" at 255,43 size 14x14
      Appearance <- "Var_VectorSecundarioJ1{7,0}"
   Circle "Circle_62" at 270,43 size 14x14
      Appearance <- "Var_VectorSecundarioJ1{7,1}"
   Circle "Circle_63" at 255,57 size 14x14
      Appearance <- "Var_VectorSecundarioJ1{7,2}"
   Circle "Circle_64" at 270,57 size 14x14
      Appearance <- "Var_VectorSecundarioJ1{7,3}"
   TextField "Text field_9" at 339,40 size 252x42; Text 'Selecciona el Codigo de tu Oponente:'
   TextField "Text field_10" at 422,20 size 67x23; Text 'INICIO'
   Circle "Circle_65" at 393,108 size 29x29
      Appearance <- "Var_CodigoSJ1{0}"
   Circle "Circle_66" at 431,107 size 29x29
      Appearance <- "Var_CodigoSJ1{1}"
   Circle "Circle_67" at 467,108 size 29x29
      Appearance <- "Var_CodigoSJ1{2}"
   Circle "Circle_68" at 505,107 size 29x29
      Appearance <- "Var_CodigoSJ1{3}"
   Button "Button_10" at 360,160 size 28x26; TextOff 'Text'
      on Press: SetBit("Panel2CafeJ1")
      on Release: SetBit("Bounce1"); ResetBit("Panel2CafeJ1")
      Appearance <- "Panel2J1Activado"
   Button "Button_11" at 392,160 size 27x26; TextOff 'Text'
      on Press: SetBit("Panel2RosaJ1")
      on Release: SetBit("Bounce1"); ResetBit("Panel2RosaJ1")
      Appearance <- "Panel2J1Activado"
   Button "Button_12" at 424,160 size 27x24; TextOff 'Text'
      on Press: SetBit("Panel2MoradoJ1")
      on Release: SetBit("Bounce1"); ResetBit("Panel2MoradoJ1")
      Appearance <- "Panel2J1Activado"
   Button "Button_13" at 458,160 size 25x25; TextOff 'Text'
      on Press: SetBit("Panel2RojoJ1")
      on Release: SetBit("Bounce1"); ResetBit("Panel2RojoJ1")
      Appearance <- "Panel2J1Activado"
   Button "Button_14" at 489,160 size 25x24; TextOff 'Text'
      on Press: SetBit("Panel2AzulJ1")
      on Release: SetBit("Bounce1"); ResetBit("Panel2AzulJ1")
      Appearance <- "Panel2J1Activado"
   Button "Button_16" at 520,160 size 25x25; TextOff 'Text'
      on Press: SetBit("Panel2VerdeJ1")
      on Release: SetBit("Bounce1"); ResetBit("Panel2VerdeJ1")
      Appearance <- "Panel2J1Activado"
   Button "Button_17" at 549,161 size 25x23; TextOff 'Text'
      on Press: SetBit("Panel2AmarilloJ1")
      on Release: SetBit("Bounce1"); ResetBit("Panel2AmarilloJ1")
      Appearance <- "Panel2J1Activado"
   Circle "Circle_69" at 342,274 size 29x29
      Appearance <- "Var_CodigoOJ1{0}"
   Circle "Circle_70" at 379,274 size 29x29
      Appearance <- "Var_CodigoOJ1{1}"
   Circle "Circle_71" at 416,274 size 29x29
      Appearance <- "Var_CodigoOJ1{2}"
   Circle "Circle_72" at 453,274 size 29x29
      Appearance <- "Var_CodigoOJ1{3}"
   TextField "Text field_11" at 341,233 size 142x23; Text 'Codigo Secreto'
   Button "Button_18" at 621,289 size 135x35; TextOff 'Reiniciar Juego'
      on Press: SetBit("ReiniciarJuego")
      on Release: ResetBit("ReiniciarJuego")
   Rectangle "Rectangle_23" at 401,90 size 13x8
      Appearance <- "Var_CodigoSJ1{0}"
   Rectangle "Rectangle_24" at 438,90 size 13x8
      Appearance <- "Var_CodigoSJ1{1}"
   Rectangle "Rectangle_25" at 475,90 size 13x8
      Appearance <- "Var_CodigoSJ1{2}"
   Rectangle "Rectangle_26" at 512,90 size 13x8
      Appearance <- "Var_CodigoSJ1{3}"
   TextField "Text field_12" at 626,28 size 120x17; Text '1. Selecciona un codigo'
      Visibility <- "Var_VectorMensajes{0}"
   TextField "Text field_13" at 627,48 size 117x43; Text '2. Esperando a que el otro jugador seleccione tu codigo'
      Visibility <- "Var_VectorMensajes{1}"
   TextField "Text field_14" at 625,94 size 130x30; Text '3. Ambos codigos seleccionados. Preparate!'
      Visibility <- "Var_VectorMensajes{2}"
   TextField "Text field_15" at 678,126 size 14x20; Text '5'
      Visibility <- "Var_VectorMensajes{3}"
   TextField "Text field_16" at 678,143 size 14x20; Text '4'
      Visibility <- "Var_VectorMensajes{4}"
   TextField "Text field_17" at 679,160 size 14x20; Text '3'
      Visibility <- "Var_VectorMensajes{5}"
   TextField "Text field_18" at 679,178 size 14x20; Text '2'
      Visibility <- "Var_VectorMensajes{6}"
   TextField "Text field_19" at 679,195 size 14x20; Text '1'
      Visibility <- "Var_VectorMensajes{7}"
   TextField "Text field_20" at 632,219 size 119x43; Text '4. Encuentra el codigo secreto antes que tu oponente!'
      Visibility <- "Var_VectorMensajes{8}"
   TextField "Text field_21" at 501,241 size 101x22; Text 'GANASTE!!!'
      Visibility <- "Var_VectorMensajes{9}"
   TextField "Text field_22" at 503,280 size 108x22; Text 'PERDISTE :('
      Visibility <- "Var_VectorMensajes{10}"

Template "Template_1" 800x442
   Button "Exit" at 720,360 size 78x58; TextOff 'Exit'; PictureOff "ExitRuntime_TP700_Comfort_TR"; PictureOn "ExitRuntime_TP700_Comfort_TR"
      on Release: StopRuntime(0)
   Button "Template_Button" at 640,360 size 78x58; TextOff 'Text'
   Button "Template_Button_1" at 560,360 size 78x58; TextOff 'Text'
   Button "Template_Button_2" at 480,360 size 78x58; TextOff 'Text'
   Button "Template_Button_3" at 400,360 size 78x58; TextOff 'Text'
   Button "Template_Button_4" at 321,360 size 78x58; TextOff 'Text'
   Button "Template_Button_5" at 241,360 size 78x58; TextOff 'Text'
   Button "Template_Button_6" at 161,360 size 78x58; TextOff 'Text'
   Button "Alarms" at 81,360 size 78x58; TextOff 'Alarms'; PictureOff "AlarmDisplay_TP700_Comfort_TR"; PictureOn "AlarmDisplay_TP700_Comfort_TR"
      on Release: function_ef3f5d25("Alarm window_Unacknowledged", -1)
   Button "Start screen" at 1,360 size 78x58; TextOff 'Start screen'; PictureOff "NavigateHome_TP700_Comfort_TR"; PictureOn "NavigateHome_TP700_Comfort_TR"
      on Release: ActivateScreen("Root screen", 0)
*)